       "PDI".CB_FLT_DC24V_K2 := "HDI_CB_FLT_DC24V_K2" XOR "IDI".CB_FLT_DC24V_K2;
       "PDI".CB_FLT_AC400V_K2 := "HDI_CB_FLT_AC400V_K2" XOR "IDI".CB_FLT_AC400V_K2;
       "PDI".SPARE_16_2 := "HDI_SPARE_16_2" XOR "IDI".SPARE_16_2;
       "PDI".CB_FLT_AC230V := "HDI_CB_FLT_AC230V" XOR "IDI".CB_FLT_AC230V;
       "PDI".SPARE_16_4 := "HDI_SPARE_16_4" XOR "IDI".SPARE_16_4;
       "PDI".SPARE_16_5 := "HDI_SPARE_16_5" XOR "IDI".SPARE_16_5;
       "PDI".SPARE_16_6 := "HDI_SPARE_16_6" XOR "IDI".SPARE_16_6;
       "PDI".SPARE_16_7 := "HDI_SPARE_16_7" XOR "IDI".SPARE_16_7;
       "PDI".SPARE_17_0 := "HDI_SPARE_17_0" XOR "IDI".SPARE_17_0;
       "PDI".UPS_24V_ALM := "HDI_UPS_24V_ALM" XOR "IDI".UPS_24V_ALM;
       "PDI".UPS_24V_NRM := "HDI_UPS_24V_NRM" XOR "IDI".UPS_24V_NRM;
       "PDI".EMO := "HDI_EMO" XOR "IDI".EMO;
       "PDI".EMS := "HDI_EMS" XOR "IDI".EMS;
       "PDI".SPARE_17_5 := "HDI_SPARE_17_5" XOR "IDI".SPARE_17_5;
       "PDI".SPARE_17_6 := "HDI_SPARE_17_6" XOR "IDI".SPARE_17_6;
       "PDI".SPARE_17_7 := "HDI_SPARE_17_7" XOR "IDI".SPARE_17_7;
       "PDI".P1_WRN := "HDI_P1_WRN" XOR "IDI".P1_WRN;
       "PDI".P1_FLT := "HDI_P1_FLT" XOR "IDI".P1_FLT;
       "PDI".P1_IS_ON := "HDI_P1_IS_ON" XOR "IDI".P1_IS_ON;
       "PDI".P1_WD := "HDI_P1_WD" XOR "IDI".P1_WD;
       "PDI".FIL_APS := "HDI_FIL_APS" XOR "IDI".FIL_APS;
       "PDI".MON_TMP_P2 := "HDI_MON_TMP_P2" XOR "IDI".MON_TMP_P2;
       "PDI".MON_TMP_P1 := "HDI_MON_TMP_P1" XOR "IDI".MON_TMP_P1;
       "PDI".SPARE_18_7 := "HDI_SPARE_18_7" XOR "IDI".SPARE_18_7;
       "PDI".FCH_LFT_SDL_NUT := "HDI_FCH_LFT_SDL_NUT" XOR "IDI".FCH_LFT_SDL_NUT;
       "PDI".LS_FCH_LFT_DN := "HDI_LS_FCH_LFT_DN" XOR "IDI".LS_FCH_LFT_DN;
       "PDI".LS_FCH_HOOK_WORK := "HDI_LS_FCH_HOOK_WORK" XOR "IDI".LS_FCH_HOOK_WORK;
       "PDI".LS_FCH_HOOK_HOME := "HDI_LS_FCH_HOOK_HOME" XOR "IDI".LS_FCH_HOOK_HOME;
       "PDI".LS_TEC_FLG_DN := "HDI_LS_TEC_FLG_DN" XOR "IDI".LS_TEC_FLG_DN;
       "PDI".TEC_FLG_SDL_NUT := "HDI_TEC_FLG_SDL_NUT" XOR "IDI".TEC_FLG_SDL_NUT;
       "PDI".LS_V11_COV_OP := "HDI_LS_V11_COV_OP" XOR "IDI".LS_V11_COV_OP;
       "PDI".LS_V11_COV_CL := "HDI_LS_V11_COV_CL" XOR "IDI".LS_V11_COV_CL;
       "PDI".GCH_APS := "HDI_GCH_APS" XOR "IDI".GCH_APS;
       "PDI".FCH_APS := "HDI_FCH_APS" XOR "IDI".FCH_APS;
       "PDI".FDR_APS := "HDI_FDR_APS" XOR "IDI".FDR_APS;
       "PDI".FIL_2_APS := "HDI_FIL_2_APS" XOR "IDI".FIL_2_APS;
       "PDI".SPARE_33_4 := "HDI_SPARE_33_4" XOR "IDI".SPARE_33_4;
       "PDI".SPARE_33_5 := "HDI_SPARE_33_5" XOR "IDI".SPARE_33_5;
       "PDI".LS_V2_1_OP := "HDI_LS_V2_1_OP" XOR "IDI".LS_V2_1_OP;
       "PDI".LS_V2_1_CL := "HDI_LS_V2_1_CL" XOR "IDI".LS_V2_1_CL;
       "PDI".CB_FLT_AC400V_K5 := "HDI_CB_FLT_AC400V_K5" XOR "IDI".CB_FLT_AC400V_K5;
       "PDI".CB_FLT_DC24V_K5 := "HDI_CB_FLT_DC24V_K5" XOR "IDI".CB_FLT_DC24V_K5;
       "PDI".LS_MAG_LFT_UP := "HDI_LS_MAG_LFT_UP" XOR "IDI".LS_MAG_LFT_UP;
       "PDI".LS_MAG_LFT_DN := "HDI_LS_MAG_LFT_DN" XOR "IDI".LS_MAG_LFT_DN;
       "PDI".SLS_MAG_LFT := "HDI_SLS_MAG_LFT" XOR "IDI".SLS_MAG_LFT;
       "PDI".MAG_LFT_SDL_NUT1 := "HDI_MAG_LFT_SDL_NUT1" XOR "IDI".MAG_LFT_SDL_NUT1;
       "PDI".MAG_LFT_SDL_NUT2 := "HDI_MAG_LFT_SDL_NUT2" XOR "IDI".MAG_LFT_SDL_NUT2;
       "PDI".MAG_LFT_SDL_NUT3 := "HDI_MAG_LFT_SDL_NUT3" XOR "IDI".MAG_LFT_SDL_NUT3;
       "PDI".OIL_LVL_CR_SFT := "HDI_OIL_LVL_CR_SFT" XOR "IDI".OIL_LVL_CR_SFT;
       "PDI".LS_V1_OP := "HDI_LS_V1_OP" XOR "IDI".LS_V1_OP;
       "PDI".LS_V1_CL := "HDI_LS_V1_CL" XOR "IDI".LS_V1_CL;
       "PDI".MP_ENB_K5 := "HDI_MP_ENB_K5" XOR "IDI".MP_ENB_K5;
       "PDI".SLS_TEC_FLG_LFT := "HDI_SLS_TEC_FLG_LFT" XOR "IDI".SLS_TEC_FLG_LFT;
       "PDI".SLS_FCH_LFT := "HDI_SLS_FCH_LFT" XOR "IDI".SLS_FCH_LFT;
       "PDI".COMP_AIR_OK := "HDI_COMP_AIR_OK" XOR "IDI".COMP_AIR_OK;
       "PDI".COMP_AIR_2_OK := "HDI_COMP_AIR_2_OK" XOR "IDI".COMP_AIR_2_OK;
       "PDI".LS_V1_1_CL := "HDI_LS_V1_1_CL" XOR "IDI".LS_V1_1_CL;
       "PDI".LS_V1_1_OP := "HDI_LS_V1_1_OP" XOR "IDI".LS_V1_1_OP;
       "PDI".LS_V3_4_OP := "HDI_LS_V3_4_OP" XOR "IDI".LS_V3_4_OP;
       "PDI".LS_V3_4_CL := "HDI_LS_V3_4_CL" XOR "IDI".LS_V3_4_CL;
       "PDI".LS_V3_3_OP := "HDI_LS_V3_3_OP" XOR "IDI".LS_V3_3_OP;
       "PDI".LS_V3_3_CL := "HDI_LS_V3_3_CL" XOR "IDI".LS_V3_3_CL;
       "PDI".LS_V2_11_OP := "HDI_LS_V2_11_OP" XOR "IDI".LS_V2_11_OP;
       "PDI".LS_V2_11_CL := "HDI_LS_V2_11_CL" XOR "IDI".LS_V2_11_CL;
       "PDI".ACC_FCH_OV_PRS_1 := "HDI_ACC_FCH_OV_PRS_1" XOR "IDI".ACC_FCH_OV_PRS_1;
       "PDI".ACC_FCH_OV_PRS_2 := "HDI_ACC_FCH_OV_PRS_2" XOR "IDI".ACC_FCH_OV_PRS_2;
       "PDI".SPARE_48_2 := "HDI_SPARE_48_2" XOR "IDI".SPARE_48_2;
       "PDI".ACC_WTR_FLW_OUT_OK := "HDI_ACC_WTR_FLW_OUT_OK" XOR "IDI".ACC_WTR_FLW_OUT_OK;
       "PDI".ACC_WTR_FLW_IN_OK := "HDI_ACC_WTR_FLW_IN_OK" XOR "IDI".ACC_WTR_FLW_IN_OK;
       "PDI".ACC_WTR_TMP_OUT_OK := "HDI_ACC_WTR_TMP_OUT_OK" XOR "IDI".ACC_WTR_TMP_OUT_OK;
       "PDI".OV_PRS_1_FLT := "HDI_OV_PRS_1_FLT" XOR "IDI".OV_PRS_1_FLT;
       "PDI".OV_PRS_2_FLT := "HDI_OV_PRS_2_FLT" XOR "IDI".OV_PRS_2_FLT;
       "PDI".ACC_SC_WTR_OK := "HDI_ACC_SC_WTR_OK" XOR "IDI".ACC_SC_WTR_OK;
       "PDI".ACC_SC_WTR_ATV := "HDI_ACC_SC_WTR_ATV" XOR "IDI".ACC_SC_WTR_ATV;
       "PDI".ACC_SC_HTR_OK := "HDI_ACC_SC_HTR_OK" XOR "IDI".ACC_SC_HTR_OK;
       "PDI".ACC_SC_HTR_ATV := "HDI_ACC_SC_HTR_ATV" XOR "IDI".ACC_SC_HTR_ATV;
       "PDI".ACC_KEY_RST := "HDI_ACC_KEY_RST" XOR "IDI".ACC_KEY_RST;
       "PDI".ACC_CB_FLT_DC24V := "HDI_ACC_CB_FLT_DC24V" XOR "IDI".ACC_CB_FLT_DC24V;
       "PDI".ACC_UPS_24V_ALM := "HDI_ACC_UPS_24V_ALM" XOR "IDI".ACC_UPS_24V_ALM;
       "PDI".ACC_UPS_24V_NRM := "HDI_ACC_UPS_24V_NRM" XOR "IDI".ACC_UPS_24V_NRM;
       "PDI".DPH_RPT_DET_OK := "HDI_DPH_RPT_DET_OK" XOR "IDI".DPH_RPT_DET_OK;
       "PDI".ACC_CB_FLT_AC230V := "HDI_ACC_CB_FLT_AC230V" XOR "IDI".ACC_CB_FLT_AC230V;
       "PDI".SPARE_90_2 := "HDI_SPARE_90_2" XOR "IDI".SPARE_90_2;
       "PDI".SPARE_90_3 := "HDI_SPARE_90_3" XOR "IDI".SPARE_90_3;
       "PDI".SPARE_90_4 := "HDI_SPARE_90_4" XOR "IDI".SPARE_90_4;
       "PDI".SPARE_90_5 := "HDI_SPARE_90_5" XOR "IDI".SPARE_90_5;
       "PDI".SPARE_90_6 := "HDI_SPARE_90_6" XOR "IDI".SPARE_90_6;
       "PDI".SPARE_90_7 := "HDI_SPARE_90_7" XOR "IDI".SPARE_90_7;
       "PDI".FU_P2_RDY := "HDI_FU_P2_RDY" XOR "IDI".FU_P2_RDY;
       "PDI".SPARE_144_1 := "HDI_SPARE_144_1" XOR "IDI".SPARE_144_1;
       "PDI".LS_GCH_UP := "HDI_LS_GCH_UP" XOR "IDI".LS_GCH_UP;
       "PDI".LS_GCH_DN := "HDI_LS_GCH_DN" XOR "IDI".LS_GCH_DN;
       "PDI".LS_GCH_SW_IN := "HDI_LS_GCH_SW_IN" XOR "IDI".LS_GCH_SW_IN;
       "PDI".LS_GCH_SW_CLN := "HDI_LS_GCH_SW_CLN" XOR "IDI".LS_GCH_SW_CLN;
       "PDI".LS_GCH_SW_OUT := "HDI_LS_GCH_SW_OUT" XOR "IDI".LS_GCH_SW_OUT;
       "PDI".LS_GCH_SW_LOCK := "HDI_LS_GCH_SW_LOCK" XOR "IDI".LS_GCH_SW_LOCK;
       "PDI".SLS_GCH_LFT := "HDI_SLS_GCH_LFT" XOR "IDI".SLS_GCH_LFT;
       "PDI".LS_TCH_UP := "HDI_LS_TCH_UP" XOR "IDI".LS_TCH_UP;
       "PDI".LS_TCH_DN := "HDI_LS_TCH_DN" XOR "IDI".LS_TCH_DN;
       "PDI".LS_TCH_SW_IN := "HDI_LS_TCH_SW_IN" XOR "IDI".LS_TCH_SW_IN;
       "PDI".LS_TCH_SW_CLN := "HDI_LS_TCH_SW_CLN" XOR "IDI".LS_TCH_SW_CLN;
       "PDI".LS_TCH_SW_OUT := "HDI_LS_TCH_SW_OUT" XOR "IDI".LS_TCH_SW_OUT;
       "PDI".LS_TCH_SW_LOCK := "HDI_LS_TCH_SW_LOCK" XOR "IDI".LS_TCH_SW_LOCK;
       "PDI".LS_TCH_TILT_0 := "HDI_LS_TCH_TILT_0" XOR "IDI".LS_TCH_TILT_0;
       "PDI".LS_TCH_TILT_30 := "HDI_LS_TCH_TILT_30" XOR "IDI".LS_TCH_TILT_30;
       "PDI".KEY_XT_LFT_SRV := "HDI_KEY_XT_LFT_SRV" XOR "IDI".KEY_XT_LFT_SRV;
       "PDI".LS_V7_UP := "HDI_LS_V7_UP" XOR "IDI".LS_V7_UP;
       "PDI".LS_V7_DN := "HDI_LS_V7_DN" XOR "IDI".LS_V7_DN;
       "PDI".LS_V7_SW_IN := "HDI_LS_V7_SW_IN" XOR "IDI".LS_V7_SW_IN;
       "PDI".LS_V7_SW_OUT := "HDI_LS_V7_SW_OUT" XOR "IDI".LS_V7_SW_OUT;
       "PDI".LS_V7_FLP_OP := "HDI_LS_V7_FLP_OP" XOR "IDI".LS_V7_FLP_OP;
       "PDI".LS_V7_CLN_POS := "HDI_LS_V7_CLN_POS" XOR "IDI".LS_V7_CLN_POS;
       "PDI".LS_GCH_BEL_UP := "HDI_LS_GCH_BEL_UP" XOR "IDI".LS_GCH_BEL_UP;
       "PDI".LS_GCH_BEL_DN := "HDI_LS_GCH_BEL_DN" XOR "IDI".LS_GCH_BEL_DN;
       "PDI".LS_XT_SLID_BW := "HDI_LS_XT_SLID_BW" XOR "IDI".LS_XT_SLID_BW;
       "PDI".LS_XT_SLID_FW := "HDI_LS_XT_SLID_FW" XOR "IDI".LS_XT_SLID_FW;
       "PDI".LS_XT_SLID_MID := "HDI_LS_XT_SLID_MID" XOR "IDI".LS_XT_SLID_MID;
       "PDI".LS_XT_CLP_CON := "HDI_LS_XT_CLP_CON" XOR "IDI".LS_XT_CLP_CON;
       "PDI".LS_XT_TILT_90 := HDI_LS_XT_TILT_90 XOR "IDI".LS_XT_TILT_90;
       "PDI".LS_XT_TILT_75 := HDI_LS_XT_TILT_75 XOR "IDI".LS_XT_TILT_75;
       "PDI".LS_UP_XT_CLP_FLT := "HDI_LS_UP_XT_CLP_FLT" XOR "IDI".LS_UP_XT_CLP_FLT;
       "PDI".SPARE_275_7 := "HDI_SPARE_275_7" XOR "IDI".SPARE_275_7;
       "PDI".LS_UP_XT_CLP_OP := "HDI_LS_UP_XT_CLP_OP" XOR "IDI".LS_UP_XT_CLP_OP;
       "PDI".LS_UP_XT_CLP_CL := "HDI_LS_UP_XT_CLP_CL" XOR "IDI".LS_UP_XT_CLP_CL;
       "PDI".LS_UP_XT_CLP_SAVE := "HDI_LS_UP_XT_CLP_SAVE" XOR "IDI".LS_UP_XT_CLP_SAVE;
       "PDI".LS_UP_XT_CLP_PLATE := "HDI_LS_UP_XT_CLP_PLATE" XOR "IDI".LS_UP_XT_CLP_PLATE;
       "PDI".LS_LO_XT_CLP_FLT := "HDI_LS_LO_XT_CLP_FLT" XOR "IDI".LS_LO_XT_CLP_FLT;
       "PDI".LS_LO_XT_CLP_OP := "HDI_LS_LO_XT_CLP_OP" XOR "IDI".LS_LO_XT_CLP_OP;
       "PDI".LS_LO_XT_CLP_CL := "HDI_LS_LO_XT_CLP_CL" XOR "IDI".LS_LO_XT_CLP_CL;
       "PDI".LS_LO_XT_CLP_SAVE := "HDI_LS_LO_XT_CLP_SAVE" XOR "IDI".LS_LO_XT_CLP_SAVE;
       "PDI".LS_LO_XT_CLP_PLATE := "HDI_LS_LO_XT_CLP_PLATE" XOR "IDI".LS_LO_XT_CLP_PLATE;
       "PDI".LS_HOI_TOOL_INST := "HDI_LS_HOI_TOOL_INST" XOR "IDI".LS_HOI_TOOL_INST;
       "PDI".XT_DRP_OUT_PRT_1_CL := "HDI_XT_DRP_OUT_PRT_1_CL" XOR "IDI".XT_DRP_OUT_PRT_1_CL;
       "PDI".XT_DRP_OUT_PRT_1_OP := "HDI_XT_DRP_OUT_PRT_1_OP" XOR "IDI".XT_DRP_OUT_PRT_1_OP;
       "PDI".XT_DRP_OUT_PRT_2_CL := "HDI_XT_DRP_OUT_PRT_2_CL" XOR "IDI".XT_DRP_OUT_PRT_2_CL;
       "PDI".XT_DRP_OUT_PRT_2_OP := "HDI_XT_DRP_OUT_PRT_2_OP" XOR "IDI".XT_DRP_OUT_PRT_2_OP;
       "PDI".CB_FLT_AC400V_K8 := "HDI_CB_FLT_AC400V_K8" XOR "IDI".CB_FLT_AC400V_K8;
       "PDI".CB_FLT_DC24V_K8 := "HDI_CB_FLT_DC24V_K8" XOR "IDI".CB_FLT_DC24V_K8;
       "PDI".XT_DRP_OUT_PRT_3_CL := "HDI_XT_DRP_OUT_PRT_3_CL" XOR "IDI".XT_DRP_OUT_PRT_3_CL;
       "PDI".XT_DRP_OUT_PRT_3_OP := "HDI_XT_DRP_OUT_PRT_3_OP" XOR "IDI".XT_DRP_OUT_PRT_3_OP;
       "PDI".XT_DRP_OUT_PRT_4_CL := "HDI_XT_DRP_OUT_PRT_4_CL" XOR "IDI".XT_DRP_OUT_PRT_4_CL;
       "PDI".XT_DRP_OUT_PRT_4_OP := "HDI_XT_DRP_OUT_PRT_4_OP" XOR "IDI".XT_DRP_OUT_PRT_4_OP;
       "PDI".LS_XT_HDL_SW_UNLOCK := "HDI_LS_XT_HDL_SW_UNLOCK" XOR "IDI".LS_XT_HDL_SW_UNLOCK;
       "PDI".LS_XT_HDL_SW_LOCK := HDI_LS_XT_HDL_SW_LOCK XOR "IDI".LS_XT_HDL_SW_LOCK;
       "PDI".LS_GCH_DOOR_OP := "HDI_LS_GCH_DOOR_OP" XOR "IDI".LS_GCH_DOOR_OP;
       "PDI".LS_GCH_DOOR_CL := "HDI_LS_GCH_DOOR_CL" XOR "IDI".LS_GCH_DOOR_CL;
       "PDI".MCC_CONTACT_XT := "HDI_MCC_CONTACT_XT" XOR "IDI".MCC_CONTACT_XT;
       "PDI".OIL_LVL_XT_SFT := "HDI_OIL_LVL_XT_SFT" XOR "IDI".OIL_LVL_XT_SFT;
       "PDI".LS_XT_SFT_SRV_POS := "HDI_LS_XT_SFT_SRV_POS" XOR "IDI".LS_XT_SFT_SRV_POS;
       "PDI".LS_XT_TOP_POS := "HDI_LS_XT_TOP_POS" XOR "IDI".LS_XT_TOP_POS;
       "PDI".SLS_TCH_LFT := "HDI_SLS_TCH_LFT" XOR "IDI".SLS_TCH_LFT;
       "PDI".XT_ROT_CAM_TRG := "HDI_XT_ROT_CAM_TRG" XOR "IDI".XT_ROT_CAM_TRG;
       "PDI".MP_ENB_K8 := "HDI_MP_ENB_K8" XOR "IDI".MP_ENB_K8;
       "PDI".MP_ENB_K9 := "HDI_MP_ENB_K9" XOR "IDI".MP_ENB_K9;
       "PDI".LS_V3_OP := "HDI_LS_V3_OP" XOR "IDI".LS_V3_OP;
       "PDI".LS_V3_CL := "HDI_LS_V3_CL" XOR "IDI".LS_V3_CL;
       "PDI".FDR_LS_V3_2_OP := "HDI_FDR_LS_V3_2_OP" XOR "IDI".FDR_LS_V3_2_OP;
       "PDI".FDR_LS_V3_2_CL := "HDI_FDR_LS_V3_2_CL" XOR "IDI".FDR_LS_V3_2_CL;
       "PDI".LSR_SEN_OBJ_DET := "HDI_LSR_SEN_OBJ_DET" XOR "IDI".LSR_SEN_OBJ_DET;
       "PDI".SPARE_280_5 := "HDI_SPARE_280_5" XOR "IDI".SPARE_280_5;
       "PDI".SPARE_280_6 := "HDI_SPARE_280_6" XOR "IDI".SPARE_280_6;
       "PDI".SPARE_280_7 := "HDI_SPARE_280_7" XOR "IDI".SPARE_280_7;
       "PDI".LS_V11_OP := "HDI_LS_V11_OP" XOR "IDI".LS_V11_OP;
       "PDI".LS_V11_CL := "HDI_LS_V11_CL" XOR "IDI".LS_V11_CL;
       "PDI".FDR_HOP_CON := "HDI_FDR_HOP_CON" XOR "IDI".FDR_HOP_CON;
   END_IF;
END_FUNCTION_BLOCK

FUNCTION_BLOCK "PM_DO"   // FB18, SCL
{ S7_Optimized_Access := 'FALSE' }
VERSION : 0.0
// --------------------------------------------------------------------------------
//     program:         PM_DO
//     description :    automatically generated PM_DO
//     name:            hp
//     date        :    03.02.2021
// 
//     revision:
//     name:
//     Date:
//                     (c)CGS
//     --------------------------------------------------------------------------------
   VAR
      y : Bool;
      count : Int := 8;
   END_VAR
   VAR_TEMP
      x : Bool;
   END_VAR
BEGIN


   IF "SY".SRM_ON THEN

       "HDO_HOR_OPP_K2" := "SDO".HOR_OPP_K2 XOR "IDO".HOR_OPP_K2;
       "HDO_LMP_RD_K2" := "SDO".LMP_RD_K2 XOR "IDO".LMP_RD_K2;
       "HDO_LMP_YE_K2" := "SDO".LMP_YE_K2 XOR "IDO".LMP_YE_K2;
       "HDO_LMP_GN_K2" := "SDO".LMP_GN_K2 XOR "IDO".LMP_GN_K2;
       "HDO_LMP_BU_K2" := "SDO".LMP_BU_K2 XOR "IDO".LMP_BU_K2;
       "HDO_HOR_MAG_ACTIVE" := "SDO".HOR_MAG_ACTIVE XOR "IDO".HOR_MAG_ACTIVE;
       "HDO_LMP_MAG_ACTIVE" := "SDO".LMP_MAG_ACTIVE XOR "IDO".LMP_MAG_ACTIVE;
       "HDO_SPARE_16_7" := "SDO".SPARE_16_7 XOR "IDO".SPARE_16_7;
       "HDO_P1_ON" := "SDO".P1_ON XOR "IDO".P1_ON;
       "HDO_P3_ON" := "SDO".P3_ON XOR "IDO".P3_ON;
       "HDO_P2_ON" := "SDO".P2_ON XOR "IDO".P2_ON;
       "HDO_P1_SEAL_GAS" := "SDO".P1_SEAL_GAS XOR "IDO".P1_SEAL_GAS;
       "HDO_P3_SEAL_GAS" := "SDO".P3_SEAL_GAS XOR "IDO".P3_SEAL_GAS;
       "HDO_HTR_PWR_ON" := "SDO".HTR_PWR_ON XOR "IDO".HTR_PWR_ON;
       "HDO_V10" := "SDO".V10 XOR "IDO".V10;
       "HDO_MON_TMP_P2_RES" := "SDO".MON_TMP_P2_RES XOR "IDO".MON_TMP_P2_RES;
       "HDO_SPARE_18_0" := "SDO".SPARE_18_0 XOR "IDO".SPARE_18_0;
       "HDO_SPARE_18_1" := "SDO".SPARE_18_1 XOR "IDO".SPARE_18_1;
       "HDO_SPARE_18_2" := "SDO".SPARE_18_2 XOR "IDO".SPARE_18_2;
       "HDO_SPARE_18_3" := "SDO".SPARE_18_3 XOR "IDO".SPARE_18_3;
       "HDO_SPARE_18_4" := "SDO".SPARE_18_4 XOR "IDO".SPARE_18_4;
       "HDO_SPARE_18_5" := "SDO".SPARE_18_5 XOR "IDO".SPARE_18_5;
       "HDO_SPARE_18_6" := "SDO".SPARE_18_6 XOR "IDO".SPARE_18_6;
       "HDO_SPARE_18_7" := "SDO".SPARE_18_7 XOR "IDO".SPARE_18_7;
       "HDO_V1_OP" := "SDO".V1_OP XOR "IDO".V1_OP;
       "HDO_V1_CL" := "SDO".V1_CL XOR "IDO".V1_CL;
       "HDO_SPARE_32_2" := "SDO".SPARE_32_2 XOR "IDO".SPARE_32_2;
       "HDO_SPARE_32_3" := "SDO".SPARE_32_3 XOR "IDO".SPARE_32_3;
       "HDO_SPARE_32_4" := "SDO".SPARE_32_4 XOR "IDO".SPARE_32_4;
       "HDO_CR_ROT_ENB" := "SDO".CR_ROT_ENB XOR "IDO".CR_ROT_ENB;
       "HDO_CR_LFT_ENB" := "SDO".CR_LFT_ENB XOR "IDO".CR_LFT_ENB;
       "HDO_FU_FCB_HDL_ON" := "SDO".FU_FCB_HDL_ON XOR "IDO".FU_FCB_HDL_ON;
       "HDO_TEC_FLG_LFT_ENB" := "SDO".TEC_FLG_LFT_ENB XOR "IDO".TEC_FLG_LFT_ENB;
       "HDO_FCH_LFT_ENB" := "SDO".FCH_LFT_ENB XOR "IDO".FCH_LFT_ENB;
       "HDO_MAG_LFT_UP" := "SDO".MAG_LFT_UP XOR "IDO".MAG_LFT_UP;
       "HDO_MAG_LFT_DN" := "SDO".MAG_LFT_DN XOR "IDO".MAG_LFT_DN;
       "HDO_BRK_MAG_LFT" := "SDO".BRK_MAG_LFT XOR "IDO".BRK_MAG_LFT;
       "HDO_SPARE_33_5" := "SDO".SPARE_33_5 XOR "IDO".SPARE_33_5;
       "HDO_SPARE_33_6" := "SDO".SPARE_33_6 XOR "IDO".SPARE_33_6;
       "HDO_SPARE_33_7" := "SDO".SPARE_33_7 XOR "IDO".SPARE_33_7;
       "HDO_V1_1_OP" := "SDO".V1_1_OP XOR "IDO".V1_1_OP;
       "HDO_V1_1_CL" := "SDO".V1_1_CL XOR "IDO".V1_1_CL;
       "HDO_SPARE_34_2" := "SDO".SPARE_34_2 XOR "IDO".SPARE_34_2;
       "HDO_SPARE_34_3" := "SDO".SPARE_34_3 XOR "IDO".SPARE_34_3;
       "HDO_SPARE_34_4" := "SDO".SPARE_34_4 XOR "IDO".SPARE_34_4;
       "HDO_SPARE_34_5" := "SDO".SPARE_34_5 XOR "IDO".SPARE_34_5;
       "HDO_SPARE_34_6" := "SDO".SPARE_34_6 XOR "IDO".SPARE_34_6;
       "HDO_SPARE_34_7" := "SDO".SPARE_34_7 XOR "IDO".SPARE_34_7;
       "HDO_ACC_SC_HTR_STR" := "SDO".ACC_SC_HTR_STR XOR "IDO".ACC_SC_HTR_STR;
       "HDO_ACC_SC_HTR_RST" := "SDO".ACC_SC_HTR_RST XOR "IDO".ACC_SC_HTR_RST;
       "HDO_ACC_SC_WTR_STR" := "SDO".ACC_SC_WTR_STR XOR "IDO".ACC_SC_WTR_STR;
       "HDO_ACC_SC_WTR_RST" := "SDO".ACC_SC_WTR_RST XOR "IDO".ACC_SC_WTR_RST;
       "HDO_ACC_ALM_LT_1" := "SDO".ACC_ALM_LT_1 XOR "IDO".ACC_ALM_LT_1;
       "HDO_ACC_ALM_SND_1" := "SDO".ACC_ALM_SND_1 XOR "IDO".ACC_ALM_SND_1;
       "HDO_ACC_ALM_LT_2" := "SDO".ACC_ALM_LT_2 XOR "IDO".ACC_ALM_LT_2;
       "HDO_ACC_ALM_SND_2" := "SDO".ACC_ALM_SND_2 XOR "IDO".ACC_ALM_SND_2;
       "HDO_FCH_HOOK_HOME" := "SDO".FCH_HOOK_HOME XOR "IDO".FCH_HOOK_HOME;
       "HDO_FCH_HOOK_WORK" := "SDO".FCH_HOOK_WORK XOR "IDO".FCH_HOOK_WORK;
       "HDO_UP_FCH_SW_BRK" := "SDO".UP_FCH_SW_BRK XOR "IDO".UP_FCH_SW_BRK;
       "HDO_LO_FCH_SW_BRK" := "SDO".LO_FCH_SW_BRK XOR "IDO".LO_FCH_SW_BRK;
       "HDO_TEC_FLG_SW_BRK" := "SDO".TEC_FLG_SW_BRK XOR "IDO".TEC_FLG_SW_BRK;
       "HDO_V25" := "SDO".V25 XOR "IDO".V25;
       "HDO_V2_1" := "SDO".V2_1 XOR "IDO".V2_1;
       "HDO_V21" := "SDO".V21 XOR "IDO".V21;
       "HDO_V19" := "SDO".V19 XOR "IDO".V19;
       "HDO_V20" := "SDO".V20 XOR "IDO".V20;
       "HDO_V22" := "SDO".V22 XOR "IDO".V22;
       "HDO_V9_2" := "SDO".V9_2 XOR "IDO".V9_2;
       "HDO_V22_1" := "SDO".V22_1 XOR "IDO".V22_1;
       "HDO_V3_4" := "SDO".V3_4 XOR "IDO".V3_4;
       "HDO_V3_3" := "SDO".V3_3 XOR "IDO".V3_3;
       "HDO_V2_11" := "SDO".V2_11 XOR "IDO".V2_11;
       "HDO_P2_FU_ON" := "SDO".P2_FU_ON XOR "IDO".P2_FU_ON;
       "HDO_P2_FU_RES" := "SDO".P2_FU_RES XOR "IDO".P2_FU_RES;
       "HDO_V4" := "SDO".V4 XOR "IDO".V4;
       "HDO_V5" := "SDO".V5 XOR "IDO".V5;
       "HDO_V6" := "SDO".V6 XOR "IDO".V6;
       "HDO_V3" := "SDO".V3 XOR "IDO".V3;
       "HDO_V3_2" := "SDO".V3_2 XOR "IDO".V3_2;
       "HDO_V24" := "SDO".V24 XOR "IDO".V24;
       "HDO_XT_DRP_OUT_PRT_CL" := "SDO".XT_DRP_OUT_PRT_CL XOR "IDO".XT_DRP_OUT_PRT_CL;
       "HDO_XT_DRP_OUT_PRT_OP" := "SDO".XT_DRP_OUT_PRT_OP XOR "IDO".XT_DRP_OUT_PRT_OP;
       "HDO_TCH_SW_LOCK" := "SDO".TCH_SW_LOCK XOR "IDO".TCH_SW_LOCK;
       "HDO_TCH_SW_UNLOCK" := "SDO".TCH_SW_UNLOCK XOR "IDO".TCH_SW_UNLOCK;
       "HDO_GCH_SW_LOCK" := "SDO".GCH_SW_LOCK XOR "IDO".GCH_SW_LOCK;
       "HDO_GCH_SW_UNLOCK" := "SDO".GCH_SW_UNLOCK XOR "IDO".GCH_SW_UNLOCK;
       "HDO_XT_HDL_SW_LOCK" := "SDO".XT_HDL_SW_LOCK XOR "IDO".XT_HDL_SW_LOCK;
       "HDO_XT_HDL_SW_UNLOCK" := "SDO".XT_HDL_SW_UNLOCK XOR "IDO".XT_HDL_SW_UNLOCK;
       "HDO_FDR_V11_OP" := "SDO".FDR_V11_OP XOR "IDO".FDR_V11_OP;
       "HDO_FDR_V11_CL" := "SDO".FDR_V11_CL XOR "IDO".FDR_V11_CL;
       "HDO_FDR_V11_CVR_OP" := "SDO".FDR_V11_CVR_OP XOR "IDO".FDR_V11_CVR_OP;
       "HDO_FDR_V11_CVR_CL" := "SDO".FDR_V11_CVR_CL XOR "IDO".FDR_V11_CVR_CL;
       "HDO_SPARE_226_2" := "SDO".SPARE_226_2 XOR "IDO".SPARE_226_2;
       "HDO_SPARE_226_3" := "SDO".SPARE_226_3 XOR "IDO".SPARE_226_3;
       "HDO_SPARE_226_4" := "SDO".SPARE_226_4 XOR "IDO".SPARE_226_4;
       "HDO_SPARE_226_5" := "SDO".SPARE_226_5 XOR "IDO".SPARE_226_5;
       "HDO_SPARE_226_6" := "SDO".SPARE_226_6 XOR "IDO".SPARE_226_6;
       "HDO_SPARE_226_7" := "SDO".SPARE_226_7 XOR "IDO".SPARE_226_7;
       "HDO_HOR_OPP_K8" := "SDO".HOR_OPP_K8 XOR "IDO".HOR_OPP_K8;
       "HDO_LMP_RD_K8" := "SDO".LMP_RD_K8 XOR "IDO".LMP_RD_K8;
       "HDO_LMP_YE_K8" := "SDO".LMP_YE_K8 XOR "IDO".LMP_YE_K8;
       "HDO_LMP_GN_K8" := "SDO".LMP_GN_K8 XOR "IDO".LMP_GN_K8;
       "HDO_LMP_BU_K8" := "SDO".LMP_BU_K8 XOR "IDO".LMP_BU_K8;
       "HDO_XT_ROT_ENB" := "SDO".XT_ROT_ENB XOR "IDO".XT_ROT_ENB;
       "HDO_XT_LFT_ENB" := "SDO".XT_LFT_ENB XOR "IDO".XT_LFT_ENB;
       "HDO_XT_HDL_LFT_ENB" := "SDO".XT_HDL_LFT_ENB XOR "IDO".XT_HDL_LFT_ENB;
       "HDO_XT_HDL_SW_ENB" := "SDO".XT_HDL_SW_ENB XOR "IDO".XT_HDL_SW_ENB;
       "HDO_FU_GCB_HDL_ON" := "SDO".FU_GCB_HDL_ON XOR "IDO".FU_GCB_HDL_ON;
       "HDO_LSR_SEN_PWR_ON" := "SDO".LSR_SEN_PWR_ON XOR "IDO".LSR_SEN_PWR_ON;
       "HDO_SPARE_273_3" := "SDO".SPARE_273_3 XOR "IDO".SPARE_273_3;
       "HDO_SPARE_273_4" := "SDO".SPARE_273_4 XOR "IDO".SPARE_273_4;
       "HDO_SPARE_273_5" := "SDO".SPARE_273_5 XOR "IDO".SPARE_273_5;
       "HDO_XT_HDL_SLID_FW" := "SDO".XT_HDL_SLID_FW XOR "IDO".XT_HDL_SLID_FW;
       "HDO_XT_HDL_SLID_BW" := "SDO".XT_HDL_SLID_BW XOR "IDO".XT_HDL_SLID_BW;
       "HDO_XT_CLP_TILT_BW" := "SDO".XT_CLP_TILT_BW XOR "IDO".XT_CLP_TILT_BW;
       "HDO_XT_CLP_TILT_FW" := "SDO".XT_CLP_TILT_FW XOR "IDO".XT_CLP_TILT_FW;
       "HDO_XT_CLP_TILT_BRK" := "SDO".XT_CLP_TILT_BRK XOR "IDO".XT_CLP_TILT_BRK;
       "HDO_XT_CLP_ABV_OP" := "SDO".XT_CLP_ABV_OP XOR "IDO".XT_CLP_ABV_OP;
       "HDO_XT_CLP_ABV_CL" := "SDO".XT_CLP_ABV_CL XOR "IDO".XT_CLP_ABV_CL;
       "HDO_XT_CLP_ABV_BRK" := "SDO".XT_CLP_ABV_BRK XOR "IDO".XT_CLP_ABV_BRK;
       "HDO_XT_CLP_ABV_RST" := "SDO".XT_CLP_ABV_RST XOR "IDO".XT_CLP_ABV_RST;
       "HDO_GCH_LFT_ENB" := "SDO".GCH_LFT_ENB XOR "IDO".GCH_LFT_ENB;
       "HDO_XT_CLP_BLW_OP" := "SDO".XT_CLP_BLW_OP XOR "IDO".XT_CLP_BLW_OP;
       "HDO_XT_CLP_BLW_CL" := "SDO".XT_CLP_BLW_CL XOR "IDO".XT_CLP_BLW_CL;
       "HDO_XT_CLP_BLW_BRK" := "SDO".XT_CLP_BLW_BRK XOR "IDO".XT_CLP_BLW_BRK;
       "HDO_XT_CLP_BLW_RST" := "SDO".XT_CLP_BLW_RST XOR "IDO".XT_CLP_BLW_RST;
       "HDO_MCC_TEST_XT" := "SDO".MCC_TEST_XT XOR "IDO".MCC_TEST_XT;
       "HDO_MCC_ENB_XT" := "SDO".MCC_ENB_XT XOR "IDO".MCC_ENB_XT;
       "HDO_TCH_LFT_ENB" := "SDO".TCH_LFT_ENB XOR "IDO".TCH_LFT_ENB;
       "HDO_TCH_TILT_ENB" := "SDO".TCH_TILT_ENB XOR "IDO".TCH_TILT_ENB;
       "HDO_GTE_V_LFT_ENB" := "SDO".GTE_V_LFT_ENB XOR "IDO".GTE_V_LFT_ENB;
       "HDO_GTE_V_SW_ENB" := "SDO".GTE_V_SW_ENB XOR "IDO".GTE_V_SW_ENB;
       "HDO_BEL_LFT_ENB" := "SDO".BEL_LFT_ENB XOR "IDO".BEL_LFT_ENB;
       "HDO_HOR_OPP_K9" := "SDO".HOR_OPP_K9 XOR "IDO".HOR_OPP_K9;
       "HDO_LMP_RD_K9" := "SDO".LMP_RD_K9 XOR "IDO".LMP_RD_K9;
       "HDO_LMP_YE_K9" := "SDO".LMP_YE_K9 XOR "IDO".LMP_YE_K9;
       "HDO_LMP_GN_K9" := "SDO".LMP_GN_K9 XOR "IDO".LMP_GN_K9;
       "HDO_LMP_BU_K9" := "SDO".LMP_BU_K9 XOR "IDO".LMP_BU_K9;
   ELSE
       IF NOT "SY".SIM_ON THEN

           "HDO_HOR_OPP_K2" := "PDO".HOR_OPP_K2 XOR "IDO".HOR_OPP_K2;
           "HDO_LMP_RD_K2" := "PDO".LMP_RD_K2 XOR "IDO".LMP_RD_K2;
           "HDO_LMP_YE_K2" := "PDO".LMP_YE_K2 XOR "IDO".LMP_YE_K2;
           "HDO_LMP_GN_K2" := "PDO".LMP_GN_K2 XOR "IDO".LMP_GN_K2;
           "HDO_LMP_BU_K2" := "PDO".LMP_BU_K2 XOR "IDO".LMP_BU_K2;
           "HDO_HOR_MAG_ACTIVE" := "PDO".HOR_MAG_ACTIVE XOR "IDO".HOR_MAG_ACTIVE;
           "HDO_LMP_MAG_ACTIVE" := "PDO".LMP_MAG_ACTIVE XOR "IDO".LMP_MAG_ACTIVE;
           "HDO_SPARE_16_7" := "PDO".SPARE_16_7 XOR "IDO".SPARE_16_7;
           "HDO_P1_ON" := "PDO".P1_ON XOR "IDO".P1_ON;
           "HDO_P3_ON" := "PDO".P3_ON XOR "IDO".P3_ON;
           "HDO_P2_ON" := "PDO".P2_ON XOR "IDO".P2_ON;
           "HDO_P1_SEAL_GAS" := "PDO".P1_SEAL_GAS XOR "IDO".P1_SEAL_GAS;
           "HDO_P3_SEAL_GAS" := "PDO".P3_SEAL_GAS XOR "IDO".P3_SEAL_GAS;
           "HDO_HTR_PWR_ON" := "PDO".HTR_PWR_ON XOR "IDO".HTR_PWR_ON;
           "HDO_V10" := "PDO".V10 XOR "IDO".V10;
           "HDO_MON_TMP_P2_RES" := "PDO".MON_TMP_P2_RES XOR "IDO".MON_TMP_P2_RES;
           "HDO_SPARE_18_0" := "PDO".SPARE_18_0 XOR "IDO".SPARE_18_0;
           "HDO_SPARE_18_1" := "PDO".SPARE_18_1 XOR "IDO".SPARE_18_1;
           "HDO_SPARE_18_2" := "PDO".SPARE_18_2 XOR "IDO".SPARE_18_2;
           "HDO_SPARE_18_3" := "PDO".SPARE_18_3 XOR "IDO".SPARE_18_3;
           "HDO_SPARE_18_4" := "PDO".SPARE_18_4 XOR "IDO".SPARE_18_4;
           "HDO_SPARE_18_5" := "PDO".SPARE_18_5 XOR "IDO".SPARE_18_5;
           "HDO_SPARE_18_6" := "PDO".SPARE_18_6 XOR "IDO".SPARE_18_6;
           "HDO_SPARE_18_7" := "PDO".SPARE_18_7 XOR "IDO".SPARE_18_7;
           "HDO_V1_OP" := "PDO".V1_OP XOR "IDO".V1_OP;
           "HDO_V1_CL" := "PDO".V1_CL XOR "IDO".V1_CL;
           "HDO_SPARE_32_2" := "PDO".SPARE_32_2 XOR "IDO".SPARE_32_2;
           "HDO_SPARE_32_3" := "PDO".SPARE_32_3 XOR "IDO".SPARE_32_3;
           "HDO_SPARE_32_4" := "PDO".SPARE_32_4 XOR "IDO".SPARE_32_4;
           "HDO_CR_ROT_ENB" := "PDO".CR_ROT_ENB XOR "IDO".CR_ROT_ENB;
           "HDO_CR_LFT_ENB" := "PDO".CR_LFT_ENB XOR "IDO".CR_LFT_ENB;
           "HDO_FU_FCB_HDL_ON" := "PDO".FU_FCB_HDL_ON XOR "IDO".FU_FCB_HDL_ON;
           "HDO_TEC_FLG_LFT_ENB" := "PDO".TEC_FLG_LFT_ENB XOR "IDO".TEC_FLG_LFT_ENB;
           "HDO_FCH_LFT_ENB" := "PDO".FCH_LFT_ENB XOR "IDO".FCH_LFT_ENB;
           "HDO_MAG_LFT_UP" := "PDO".MAG_LFT_UP XOR "IDO".MAG_LFT_UP;
           "HDO_MAG_LFT_DN" := "PDO".MAG_LFT_DN XOR "IDO".MAG_LFT_DN;
           "HDO_BRK_MAG_LFT" := "PDO".BRK_MAG_LFT XOR "IDO".BRK_MAG_LFT;
           "HDO_SPARE_33_5" := "PDO".SPARE_33_5 XOR "IDO".SPARE_33_5;
           "HDO_SPARE_33_6" := "PDO".SPARE_33_6 XOR "IDO".SPARE_33_6;
           "HDO_SPARE_33_7" := "PDO".SPARE_33_7 XOR "IDO".SPARE_33_7;
           "HDO_V1_1_OP" := "PDO".V1_1_OP XOR "IDO".V1_1_OP;
           "HDO_V1_1_CL" := "PDO".V1_1_CL XOR "IDO".V1_1_CL;
           "HDO_SPARE_34_2" := "PDO".SPARE_34_2 XOR "IDO".SPARE_34_2;
           "HDO_SPARE_34_3" := "PDO".SPARE_34_3 XOR "IDO".SPARE_34_3;
           "HDO_SPARE_34_4" := "PDO".SPARE_34_4 XOR "IDO".SPARE_34_4;
           "HDO_SPARE_34_5" := "PDO".SPARE_34_5 XOR "IDO".SPARE_34_5;
           "HDO_SPARE_34_6" := "PDO".SPARE_34_6 XOR "IDO".SPARE_34_6;
           "HDO_SPARE_34_7" := "PDO".SPARE_34_7 XOR "IDO".SPARE_34_7;
           "HDO_ACC_SC_HTR_STR" := "PDO".ACC_SC_HTR_STR XOR "IDO".ACC_SC_HTR_STR;
           "HDO_ACC_SC_HTR_RST" := "PDO".ACC_SC_HTR_RST XOR "IDO".ACC_SC_HTR_RST;
           "HDO_ACC_SC_WTR_STR" := "PDO".ACC_SC_WTR_STR XOR "IDO".ACC_SC_WTR_STR;
           "HDO_ACC_SC_WTR_RST" := "PDO".ACC_SC_WTR_RST XOR "IDO".ACC_SC_WTR_RST;
           "HDO_ACC_ALM_LT_1" := "PDO".ACC_ALM_LT_1 XOR "IDO".ACC_ALM_LT_1;
           "HDO_ACC_ALM_SND_1" := "PDO".ACC_ALM_SND_1 XOR "IDO".ACC_ALM_SND_1;
           "HDO_ACC_ALM_LT_2" := "PDO".ACC_ALM_LT_2 XOR "IDO".ACC_ALM_LT_2;
           "HDO_ACC_ALM_SND_2" := "PDO".ACC_ALM_SND_2 XOR "IDO".ACC_ALM_SND_2;
           "HDO_FCH_HOOK_HOME" := "PDO".FCH_HOOK_HOME XOR "IDO".FCH_HOOK_HOME;
           "HDO_FCH_HOOK_WORK" := "PDO".FCH_HOOK_WORK XOR "IDO".FCH_HOOK_WORK;
           "HDO_UP_FCH_SW_BRK" := "PDO".UP_FCH_SW_BRK XOR "IDO".UP_FCH_SW_BRK;
           "HDO_LO_FCH_SW_BRK" := "PDO".LO_FCH_SW_BRK XOR "IDO".LO_FCH_SW_BRK;
           "HDO_TEC_FLG_SW_BRK" := "PDO".TEC_FLG_SW_BRK XOR "IDO".TEC_FLG_SW_BRK;
           "HDO_V25" := "PDO".V25 XOR "IDO".V25;
           "HDO_V2_1" := "PDO".V2_1 XOR "IDO".V2_1;
           "HDO_V21" := "PDO".V21 XOR "IDO".V21;
           "HDO_V19" := "PDO".V19 XOR "IDO".V19;
           "HDO_V20" := "PDO".V20 XOR "IDO".V20;
           "HDO_V22" := "PDO".V22 XOR "IDO".V22;
           "HDO_V9_2" := "PDO".V9_2 XOR "IDO".V9_2;
           "HDO_V22_1" := "PDO".V22_1 XOR "IDO".V22_1;
           "HDO_V3_4" := "PDO".V3_4 XOR "IDO".V3_4;
           "HDO_V3_3" := "PDO".V3_3 XOR "IDO".V3_3;
           "HDO_V2_11" := "PDO".V2_11 XOR "IDO".V2_11;
           "HDO_P2_FU_ON" := "PDO".P2_FU_ON XOR "IDO".P2_FU_ON;
           "HDO_P2_FU_RES" := "PDO".P2_FU_RES XOR "IDO".P2_FU_RES;
           "HDO_V4" := "PDO".V4 XOR "IDO".V4;
           "HDO_V5" := "PDO".V5 XOR "IDO".V5;
           "HDO_V6" := "PDO".V6 XOR "IDO".V6;
           "HDO_V3" := "PDO".V3 XOR "IDO".V3;
           "HDO_V3_2" := "PDO".V3_2 XOR "IDO".V3_2;
           "HDO_V24" := "PDO".V24 XOR "IDO".V24;
           "HDO_XT_DRP_OUT_PRT_CL" := "PDO".XT_DRP_OUT_PRT_CL XOR "IDO".XT_DRP_OUT_PRT_CL;
           "HDO_XT_DRP_OUT_PRT_OP" := "PDO".XT_DRP_OUT_PRT_OP XOR "IDO".XT_DRP_OUT_PRT_OP;
           "HDO_TCH_SW_LOCK" := "PDO".TCH_SW_LOCK XOR "IDO".TCH_SW_LOCK;
           "HDO_TCH_SW_UNLOCK" := "PDO".TCH_SW_UNLOCK XOR "IDO".TCH_SW_UNLOCK;
           "HDO_GCH_SW_LOCK" := "PDO".GCH_SW_LOCK XOR "IDO".GCH_SW_LOCK;
           "HDO_GCH_SW_UNLOCK" := "PDO".GCH_SW_UNLOCK XOR "IDO".GCH_SW_UNLOCK;
           "HDO_XT_HDL_SW_LOCK" := "PDO".XT_HDL_SW_LOCK XOR "IDO".XT_HDL_SW_LOCK;
           "HDO_XT_HDL_SW_UNLOCK" := "PDO".XT_HDL_SW_UNLOCK XOR "IDO".XT_HDL_SW_UNLOCK;
           "HDO_FDR_V11_OP" := "PDO".FDR_V11_OP XOR "IDO".FDR_V11_OP;
           "HDO_FDR_V11_CL" := "PDO".FDR_V11_CL XOR "IDO".FDR_V11_CL;
           "HDO_FDR_V11_CVR_OP" := "PDO".FDR_V11_CVR_OP XOR "IDO".FDR_V11_CVR_OP;
           "HDO_FDR_V11_CVR_CL" := "PDO".FDR_V11_CVR_CL XOR "IDO".FDR_V11_CVR_CL;
           "HDO_SPARE_226_2" := "PDO".SPARE_226_2 XOR "IDO".SPARE_226_2;
           "HDO_SPARE_226_3" := "PDO".SPARE_226_3 XOR "IDO".SPARE_226_3;
           "HDO_SPARE_226_4" := "PDO".SPARE_226_4 XOR "IDO".SPARE_226_4;
           "HDO_SPARE_226_5" := "PDO".SPARE_226_5 XOR "IDO".SPARE_226_5;
           "HDO_SPARE_226_6" := "PDO".SPARE_226_6 XOR "IDO".SPARE_226_6;
           "HDO_SPARE_226_7" := "PDO".SPARE_226_7 XOR "IDO".SPARE_226_7;
           "HDO_HOR_OPP_K8" := "PDO".HOR_OPP_K8 XOR "IDO".HOR_OPP_K8;
           "HDO_LMP_RD_K8" := "PDO".LMP_RD_K8 XOR "IDO".LMP_RD_K8;
           "HDO_LMP_YE_K8" := "PDO".LMP_YE_K8 XOR "IDO".LMP_YE_K8;
           "HDO_LMP_GN_K8" := "PDO".LMP_GN_K8 XOR "IDO".LMP_GN_K8;
           "HDO_LMP_BU_K8" := "PDO".LMP_BU_K8 XOR "IDO".LMP_BU_K8;
           "HDO_XT_ROT_ENB" := "PDO".XT_ROT_ENB XOR "IDO".XT_ROT_ENB;
           "HDO_XT_LFT_ENB" := "PDO".XT_LFT_ENB XOR "IDO".XT_LFT_ENB;
           "HDO_XT_HDL_LFT_ENB" := "PDO".XT_HDL_LFT_ENB XOR "IDO".XT_HDL_LFT_ENB;
           "HDO_XT_HDL_SW_ENB" := "PDO".XT_HDL_SW_ENB XOR "IDO".XT_HDL_SW_ENB;
           "HDO_FU_GCB_HDL_ON" := "PDO".FU_GCB_HDL_ON XOR "IDO".FU_GCB_HDL_ON;
           "HDO_LSR_SEN_PWR_ON" := "PDO".LSR_SEN_PWR_ON XOR "IDO".LSR_SEN_PWR_ON;
           "HDO_SPARE_273_3" := "PDO".SPARE_273_3 XOR "IDO".SPARE_273_3;
           "HDO_SPARE_273_4" := "PDO".SPARE_273_4 XOR "IDO".SPARE_273_4;
           "HDO_SPARE_273_5" := "PDO".SPARE_273_5 XOR "IDO".SPARE_273_5;
           "HDO_XT_HDL_SLID_FW" := "PDO".XT_HDL_SLID_FW XOR "IDO".XT_HDL_SLID_FW;
           "HDO_XT_HDL_SLID_BW" := "PDO".XT_HDL_SLID_BW XOR "IDO".XT_HDL_SLID_BW;
           "HDO_XT_CLP_TILT_BW" := "PDO".XT_CLP_TILT_BW XOR "IDO".XT_CLP_TILT_BW;
           "HDO_XT_CLP_TILT_FW" := "PDO".XT_CLP_TILT_FW XOR "IDO".XT_CLP_TILT_FW;
           "HDO_XT_CLP_TILT_BRK" := "PDO".XT_CLP_TILT_BRK XOR "IDO".XT_CLP_TILT_BRK;
           "HDO_XT_CLP_ABV_OP" := "PDO".XT_CLP_ABV_OP XOR "IDO".XT_CLP_ABV_OP;
           "HDO_XT_CLP_ABV_CL" := "PDO".XT_CLP_ABV_CL XOR "IDO".XT_CLP_ABV_CL;
           "HDO_XT_CLP_ABV_BRK" := "PDO".XT_CLP_ABV_BRK XOR "IDO".XT_CLP_ABV_BRK;
           "HDO_XT_CLP_ABV_RST" := "PDO".XT_CLP_ABV_RST XOR "IDO".XT_CLP_ABV_RST;
           "HDO_GCH_LFT_ENB" := "PDO".GCH_LFT_ENB XOR "IDO".GCH_LFT_ENB;
           "HDO_XT_CLP_BLW_OP" := "PDO".XT_CLP_BLW_OP XOR "IDO".XT_CLP_BLW_OP;
           "HDO_XT_CLP_BLW_CL" := "PDO".XT_CLP_BLW_CL XOR "IDO".XT_CLP_BLW_CL;
           "HDO_XT_CLP_BLW_BRK" := "PDO".XT_CLP_BLW_BRK XOR "IDO".XT_CLP_BLW_BRK;
           "HDO_XT_CLP_BLW_RST" := "PDO".XT_CLP_BLW_RST XOR "IDO".XT_CLP_BLW_RST;
           "HDO_MCC_TEST_XT" := "PDO".MCC_TEST_XT XOR "IDO".MCC_TEST_XT;
           "HDO_MCC_ENB_XT" := "PDO".MCC_ENB_XT XOR "IDO".MCC_ENB_XT;
           "HDO_TCH_LFT_ENB" := "PDO".TCH_LFT_ENB XOR "IDO".TCH_LFT_ENB;
           "HDO_TCH_TILT_ENB" := "PDO".TCH_TILT_ENB XOR "IDO".TCH_TILT_ENB;
           "HDO_GTE_V_LFT_ENB" := "PDO".GTE_V_LFT_ENB XOR "IDO".GTE_V_LFT_ENB;
           "HDO_GTE_V_SW_ENB" := "PDO".GTE_V_SW_ENB XOR "IDO".GTE_V_SW_ENB;
           "HDO_BEL_LFT_ENB" := "PDO".BEL_LFT_ENB XOR "IDO".BEL_LFT_ENB;
           "HDO_HOR_OPP_K9" := "PDO".HOR_OPP_K9 XOR "IDO".HOR_OPP_K9;
           "HDO_LMP_RD_K9" := "PDO".LMP_RD_K9 XOR "IDO".LMP_RD_K9;
           "HDO_LMP_YE_K9" := "PDO".LMP_YE_K9 XOR "IDO".LMP_YE_K9;
           "HDO_LMP_GN_K9" := "PDO".LMP_GN_K9 XOR "IDO".LMP_GN_K9;
           "HDO_LMP_BU_K9" := "PDO".LMP_BU_K9 XOR "IDO".LMP_BU_K9;
       END_IF;
   END_IF;
END_FUNCTION_BLOCK

FUNCTION_BLOCK "PM_AI"   // FB19, SCL
{ S7_Optimized_Access := 'FALSE' }
VERSION : 0.0
// --------------------------------------------------------------------------------
//     program:         PM_AI
//     description :    automatically generated PM_AI
//     name:            hp
//     date        :    03.02.2021
// 
//     revision:
//     name:
//     Date:
//                     (c)CGS
//     --------------------------------------------------------------------------------
   VAR
      y : Bool;
      count : Int := 8;
   END_VAR
   VAR_TEMP
      x : Bool;
   END_VAR
BEGIN


   IF "SY".SIM_ON AND NOT "SY".SRM_ON THEN

       "PAI".TRV_ACT_POS := "SAI".TRV_ACT_POS;
       "PAI".TRV_ACT_POS_1 := "SAI".TRV_ACT_POS_1;
       "PAI".TRV_PRS_FIL_1 := "SAI".TRV_PRS_FIL_1;
       "PAI".TRV_PRS_FIL_2 := "SAI".TRV_PRS_FIL_2;
       "PAI".PYR_ACT_HTR_1_TMP := "SAI".PYR_ACT_HTR_1_TMP;
       "PAI".ACT_PRS_AR_VSL := "SAI".ACT_PRS_AR_VSL;
       "PAI".PYR_ACT_MELT_TMP := "SAI".PYR_ACT_MELT_TMP;
       "PAI".GCH_PCR_ACT_PRS := "SAI".GCH_PCR_ACT_PRS;
       "PAI".FCH_PCR_ACT_PRS := "SAI".FCH_PCR_ACT_PRS;
       "PAI".FCH_BAR_ACT_PRS_100 := "SAI".FCH_BAR_ACT_PRS_100;
       "PAI".ACC_WTR_TMP := "SAI".ACC_WTR_TMP;
       "PAI".ACC_WTR_PRS_IN := "SAI".ACC_WTR_PRS_IN;
       "PAI".ACC_WTR_FLW_OUT := "SAI".ACC_WTR_FLW_OUT;
       "PAI".ACC_WTR_FLW_IN := "SAI".ACC_WTR_FLW_IN;
       "PAI".ACC_WTR_SPL_PRS := "SAI".ACC_WTR_SPL_PRS;
       "PAI".ACC_SPARE_810 := "SAI".ACC_SPARE_810;
   ELSE

       "PAI".TRV_ACT_POS := "PM_AI_CONVERT" (CHANNEL := "HAI".TRV_ACT_POS, CONVERT_PAR:="CAI".CONFIG_DATA[1]);
       "PAI".TRV_ACT_POS_1 := "PM_AI_CONVERT" (CHANNEL := "HAI".TRV_ACT_POS_1, CONVERT_PAR:="CAI".CONFIG_DATA[2]);
       "PAI".TRV_PRS_FIL_1 := "PM_AI_CONVERT" (CHANNEL := "HAI".TRV_PRS_FIL_1, CONVERT_PAR:="CAI".CONFIG_DATA[3]);
       "PAI".TRV_PRS_FIL_2 := "PM_AI_CONVERT" (CHANNEL := "HAI".TRV_PRS_FIL_2, CONVERT_PAR:="CAI".CONFIG_DATA[4]);
       "PAI".PYR_ACT_HTR_1_TMP := "PM_AI_CONVERT" (CHANNEL := "HAI".PYR_ACT_HTR_1_TMP, CONVERT_PAR:="CAI".CONFIG_DATA[5]);
       "PAI".ACT_PRS_AR_VSL := "PM_AI_CONVERT" (CHANNEL := "HAI".ACT_PRS_AR_VSL, CONVERT_PAR:="CAI".CONFIG_DATA[6]);
       "PAI".PYR_ACT_MELT_TMP := "PM_AI_CONVERT" (CHANNEL := "HAI".PYR_ACT_MELT_TMP, CONVERT_PAR:="CAI".CONFIG_DATA[7]);
       "PAI".GCH_PCR_ACT_PRS := "PM_AI_CONVERT" (CHANNEL := "HAI".GCH_PCR_ACT_PRS, CONVERT_PAR:="CAI".CONFIG_DATA[8]);
       "PAI".FCH_PCR_ACT_PRS := "PM_AI_CONVERT" (CHANNEL := "HAI".FCH_PCR_ACT_PRS, CONVERT_PAR:="CAI".CONFIG_DATA[9]);
       "PAI".FCH_BAR_ACT_PRS_100 := "PM_AI_CONVERT" (CHANNEL := "HAI".FCH_BAR_ACT_PRS_100, CONVERT_PAR:="CAI".CONFIG_DATA[10]);
       "PAI".ACC_WTR_TMP := "PM_AI_CONVERT" (CHANNEL := "HAI".ACC_WTR_TMP, CONVERT_PAR:="CAI".CONFIG_DATA[11]);
       "PAI".ACC_WTR_PRS_IN := "PM_AI_CONVERT" (CHANNEL := "HAI".ACC_WTR_PRS_IN, CONVERT_PAR:="CAI".CONFIG_DATA[12]);
       "PAI".ACC_WTR_FLW_OUT := "PM_AI_CONVERT" (CHANNEL := "HAI".ACC_WTR_FLW_OUT, CONVERT_PAR:="CAI".CONFIG_DATA[13]);
       "PAI".ACC_WTR_FLW_IN := "PM_AI_CONVERT" (CHANNEL := "HAI".ACC_WTR_FLW_IN, CONVERT_PAR:="CAI".CONFIG_DATA[14]);
       "PAI".ACC_WTR_SPL_PRS := "PM_AI_CONVERT" (CHANNEL := "HAI".ACC_WTR_SPL_PRS, CONVERT_PAR:="CAI".CONFIG_DATA[15]);
       "PAI".ACC_SPARE_810 := "PM_AI_CONVERT" (CHANNEL := "HAI".ACC_SPARE_810, CONVERT_PAR:="CAI".CONFIG_DATA[16]);
   END_IF;
END_FUNCTION_BLOCK

FUNCTION_BLOCK "PM_AO"   // FB20, SCL
{ S7_Optimized_Access := 'FALSE' }
VERSION : 0.0
// --------------------------------------------------------------------------------
//     program:         PM_AO
//     description :    automatically generated PM_AO
//     name:            hp
//     date        :    03.02.2021
// 
//     revision:
//     name:
//     Date:
//                     (c)CGS
//     --------------------------------------------------------------------------------
   VAR
      y : Bool;
      count : Int := 8;
   END_VAR
   VAR_TEMP
      x : Bool;
   END_VAR
BEGIN


   IF "SY".SRM_ON THEN

       "HAO".TRV_SET_POS := "PM_AO_CONVERT"(OUTVALUE := "SAO".TRV_SET_POS, CONVERT_PAR := "CAO".CONFIG_DATA[1]);
       "HAO".TRV_SET_POS_1 := "PM_AO_CONVERT"(OUTVALUE := "SAO".TRV_SET_POS_1, CONVERT_PAR := "CAO".CONFIG_DATA[2]);
   ELSE
       IF NOT "SY".SIM_ON THEN

           "HAO".TRV_SET_POS := "PM_AO_CONVERT"(OUTVALUE := "PAO".TRV_SET_POS, CONVERT_PAR := "CAO".CONFIG_DATA[1]);
           "HAO".TRV_SET_POS_1 := "PM_AO_CONVERT"(OUTVALUE := "PAO".TRV_SET_POS_1, CONVERT_PAR := "CAO".CONFIG_DATA[2]);
       END_IF;
   END_IF;
END_FUNCTION_BLOCK

FUNCTION_BLOCK "PM_GET_WGT_XT_CLP"   // FB29, SCL
{ S7_Optimized_Access := 'FALSE' }
VERSION : 0.0
// --------------------------------------------------------------------------------
//     program     :    PM_GET_WGT_XT_CLP
//     description :    read load cell data and convert in weight unit   
//     name        :    lv
//     date        :    21.09.2016
// 
//     revision    :    
//     name        :
//     date        :    
//                     (c)CGS
//     --------------------------------------------------------------------------------
   VAR
      i : Int;
      bdg_vlt_clp_wgt : Real;   // bridge voltage load cell
      ref_vlt_clp_wgt : Real;   // reference voltage load cell
      start_si_lvl : Real;
      mess_si_lvl : Real;
      hop_cone : Real;
      hop_cute : Real;
      hop_cyl_start : Real;
      hop_cyl_mess : Real;
      hop_sum : Real;
      hop_mess : Real;
      tar_xt_clp_wgt : Bool;
      fl_tar_xt_clp_wgt : Bool;
   END_VAR
   VAR_TEMP
      Kl3351_1_IN : Struct
         D1_0 : Byte;   // High byte channel 1
         D0_0 : Byte;   // Low byte channel 1
         D1_1 : Byte;   // High byte channel 2
         D0_1 : Byte;   // Low byte channel 2
      END_STRUCT;
      Kl3351_1_OUT : Struct
         D1_0 : Byte;   // High byte channel 1
         D0_0 : Byte;   // Low byte channel 1
         D1_1 : Byte;   // High byte channel 2
         D0_1 : Byte;   // Low byte channel 2
      END_STRUCT;
      Dprd_RetVal_1 : Int;
      data_int : Int;
      data_word : Word;
      ctrl_byte : Byte;
      lb_data_word : Byte;
      hb_data_word : Byte;
   END_VAR
   VAR CONSTANT
      bdg_vlt_sca_fct : Real := 5.0E-07;   // bridge voltage scaling factor (500nV/digit) siehe Beckhoff Doku
      ref_vlt_sca_fct : Real := 0.0005;   // reference voltage scaling factor (500yV/digit) siehe Beckhoff Doku
      rtd_val_clp_wgt_cell : Real := 2.0E-05;   // 2 mV/V rated characteristic value crystal weight load cell
   END_VAR
BEGIN

       //---------------------------
       //read out process data feeder load cell
       //----------------------------------------------
       #Dprd_RetVal_1         := DPRD_DAT(LADDR :=  16#610,            //addr: 1552
                                           RECORD =>  #Kl3351_1_IN);
       //channel one
       //-----------
       //sta_byte_1          :=  Kl3351_1_IN.ST_0;  
       #lb_data_word        :=  #Kl3351_1_IN.D0_0;
       #hb_data_word        :=  #Kl3351_1_IN.D1_0;

       #data_word           :=  SHL(IN:=BYTE_TO_WORD(#hb_data_word), N:=8) OR BYTE_TO_WORD(#lb_data_word);
       #data_int            :=  WORD_TO_INT(#data_word);

       #bdg_vlt_clp_wgt          := (INT_TO_REAL(#data_int)) * #bdg_vlt_sca_fct;

       //channel two
       //-----------
       //sta_byte_2          :=  Kl3351_1_IN.ST_1;  
       #lb_data_word        :=  #Kl3351_1_IN.D0_1;
       #hb_data_word        :=  #Kl3351_1_IN.D1_1;

       #data_word           :=  SHL(IN:=BYTE_TO_WORD(#hb_data_word), N:=8) OR BYTE_TO_WORD(#lb_data_word);
       #data_int            :=  WORD_TO_INT(#data_word);

       #ref_vlt_clp_wgt     := (INT_TO_REAL(#data_int)) * #ref_vlt_sca_fct;


       //calculation of feeder cute weight in g
       //----------------------------------
       IF NOT "SY".SIM_ON    THEN                //simulation mode disabled?
           IF (#ref_vlt_clp_wgt > 0.0)   THEN 
               "AV".XT_HDL_CLP_WGT  := ((#bdg_vlt_clp_wgt / #ref_vlt_clp_wgt) * (10.0 / #rtd_val_clp_wgt_cell)) 
                                         * "CNF".XT_CLP_LDC_CAL;

           END_IF;
       END_IF;

      IF "PDI".LS_XT_CLP_CON THEN               // create auto calibration bit
         IF ("DIS".ACT_POS_XT_HDL_LFT>400.0) AND NOT "LT".XT_HDL_LFT_UP AND NOT "LT".XT_HDL_LFT_DN AND NOT #fl_tar_xt_clp_wgt THEN 
            #tar_xt_clp_wgt    := True;
            #fl_tar_xt_clp_wgt := True;
         END_IF;
      ELSE
         #tar_xt_clp_wgt    := false;
         #fl_tar_xt_clp_wgt := false;
      END_IF;        

       //set display variable
       //--------------------
       IF "PDI".LS_XT_CLP_CON OR "SysLog1" THEN
           "DIS".XT_HDL_CLP_WGT      :=  "AV".XT_HDL_CLP_WGT;   
           "DIS".XT_HDL_CLP_WGT_TAR  :=  "AV".XT_HDL_CLP_WGT - "AV".XT_HDL_CLP_TAR_WGT;
           IF "CNF".XT_CLP_LDC_CAL= 0.0 THEN
              "CNF".XT_CLP_LDC_CAL := 1.0;
           END_IF;
           IF ("KYD".XT_CLP_WGT_TAR) OR #tar_xt_clp_wgt THEN
               "AV".XT_HDL_CLP_TAR_WGT := "AV".XT_HDL_CLP_WGT;
               #tar_xt_clp_wgt := false;
           END_IF;     
       ELSE
           "DIS".XT_HDL_CLP_WGT      :=  0.0;   
           "DIS".XT_HDL_CLP_WGT_TAR  :=  0.0;
           "AV".XT_HDL_CLP_WGT       :=  0.0;   
           "AV".XT_HDL_CLP_TAR_WGT   :=  0.0;
       END_IF;
END_FUNCTION_BLOCK

FUNCTION_BLOCK "PM_TLU_PWR_SPL"   // FB33, SCL
{ S7_Optimized_Access := 'FALSE' }
VERSION : 0.0
// --------------------------------------------------------------------------------
//     program     :   PM_TLU_PWR_SPL  
//     description :   data transfer from and to TLU power supply profibus module
//     name        :   G. Eibelsh鋟ser  
//     date        :   16.04.2012
// 
//     revision    :
//     name        :
//     DATE        :    
//                     (c) PVATepla AG
//     --------------------------------------------------------------------------------
   VAR_INPUT
      htr_enb : Bool;   // heater enable
      htr_rst : Bool;   // heater reset
      fst_byte_offs : Int;   // first record byte in DB PM_TLU_PWR_SPL_DATA_BUF
      dp_adress : Word;   // address to read/write data from/to (DP Adress ID LADDR)
      set_htr_pwr : Real;
      htr_pwr_rng : Real;
      htr_cur_rng : Real;
      htr_vlt_rng : Real;
   END_VAR
   VAR_OUTPUT
      sta_htr_on : Bool;
      sta_error : Bool;
      sta_warn : Bool;
      sta_pi_mode : Bool;
      sta_pu_mode : Bool;
      sta_i_mode : Bool;
      sta_u_mode : Bool;
      sta_saved : Bool;
      flt_i_pri : Bool;
      flt_i_max : Bool;
      flt_u_max : Bool;
      flt_wire : Bool;
      flt_flash : Bool;
      flt_trafo : Bool;
      flt_data_flow : Bool;
      flt_data_com : Bool;
      flt_data : Bool;
      flt_tast : Bool;
      flt_ua_max : Bool;
      flt_u_min : Bool;
      flt_temp : Bool;
      flt_sense : Bool;
      flt_igbt : Bool;
      flt_dioden : Bool;
      flt_3 : Bool;
      flt_shunt : Bool;
      flt_board : Bool;
      flt_6 : Bool;
      flt_soft : Bool;
      flt_timeout : Bool;
      flt_short : Bool;
      act_htr_cur : Real;
      act_htr_vlt : Real;
      act_htr_pwr : Real;
   END_VAR
   VAR
      htr_word_sta_1 : Word;
      htr_word_flt_1 : Word;
      htr_word_flt_2 : Word;
      htr_word_flt_mem_1 : Word;
      htr_word_flt_mem_2 : Word;
      htr_word_cur_n : Word;
      htr_word_vlt_n : Word;
      htr_word_pwr_n : Word;
      htr_word_sta_2 : Word;
      htr_word_enrj_1 : Word;
      htr_word_enrj_2 : Word;
      htr_word_enrj_3 : Word;
      htr_word_pls : Word;
      htr_word_presc : Word;
      htr_word_firm : Word;
   END_VAR
   VAR_TEMP
      Buffer : "UDT_ANY_POINTER";
      Temp_Any_Pointer AT Buffer : ANY;
      RetVal : Int;   // Return Value of SFC 14/15
      DB_Byte_Adr : Int;   // start address in DB for reading/writing
      ctrl_low_byte : Byte;
      ctrl_high_byte : Byte;
      ctrl_word : Word;
      set_pwr_word : Word;
      set_cur_word : Word;
      set_vlt_word : Word;
      htr_word_cur : Word;
      htr_word_vlt : Word;
      htr_word_pwr : Word;
      set_pwr : Real;
      set_cur : Real;
      set_vlt : Real;
   END_VAR
   VAR CONSTANT
      DB_Number : Int := 127;   // number of buffer data block containing data of SFC 14/15
      Byte_Count : Int := 6;   // number of bytes to read/write consistently
      res : Int := 25000;   // resolution of TLU data
   END_VAR
BEGIN

       //preset values for 10 Byte Buffer for ANY_Pointer 
       //------------------------------------------------
       #Buffer.Syntax_Id := B#16#10;    // buffer length - MUST always be 16#10! (S7 needs 10 bytes to save the data of...
                                       // ...parameter of type 'ANY')                                                
       #Buffer.DataType := B#16#02;     // code f黵 data type 'BYTE'

       (************************************************************************************************************* 
          code for data types:
          --------------------
           b#16#00 = NIL,      b#16#01 = BOOL,     b#16#02 = BYTE,     b#16#03 = CHAR,     b#16#04 = WORD, b#16#05 = INT, 
           b#16#06 = DWORD,    b#16#07 = DINT,     b#16#08 = REAL,     b#16#09 = DATE,     b#16#0A = TIME_OF_DAY (TOD), 
           b#16#0B = TIME,     b#16#0C = S5TIME,   b#16#0E = DATE_AND_TIME (DT),           b#16#13 = STRING            
       **************************************************************************************************************) 

       #Buffer.Count        := INT_TO_WORD(32);          // number of bytes to read
       #Buffer.DB_Number    := INT_TO_WORD(#DB_Number);  
       (********************************************************************************** 
          code for memory area (=> highest byte of Buffer.Byte_Pointer)
          --------------------
           b#16#81 = E,    b#16#82 = A,    b#16#83 = M,    b#16#84 = DB,   b#16#85 = DI,
           b#16#86 = L,    b#16#87 = V
       ***********************************************************************************)
       //read the first Byte Block data from Plating profibus module Byte 0..31
       //----------------------------------
       #Buffer.Byte_Pointer := DW#16#8400_0000;                             // Null Pointer to global data DBX0.0 (code for memory data)
       #DB_Byte_Adr := #fst_byte_offs;                                       //set start byte address in DB PM_TLU_PWR_SPL_DATA_BUF for reading
       #Buffer.Byte_Pointer := #Buffer.Byte_Pointer OR (SHL(IN:=WORD_TO_DWORD(INT_TO_WORD(#DB_Byte_Adr)),N:=3));  // bits 0..2 of Byte_Pointer contain bit-add         
       #RetVal := DPRD_DAT(LADDR:= #dp_adress, RECORD=>#Temp_Any_Pointer);    // read values from periphery
       //---------------------------------------------------------------------------------------------------------------------

       //read the second Byte Block data from Plating profibus module 32..35
       #Buffer.Count        := INT_TO_WORD(4);          // number of bytes to read
       #Buffer.DB_Number    := INT_TO_WORD(#DB_Number);  

       (********************************************************************************** 
          code for memory area (=> highest byte of Buffer.Byte_Pointer)
          --------------------
           b#16#81 = E,    b#16#82 = A,    b#16#83 = M,    b#16#84 = DB,   b#16#85 = DI,
           b#16#86 = L,    b#16#87 = V
       ***********************************************************************************) 
       //----------------------------------
       #Buffer.Byte_Pointer := DW#16#8400_0000;                             // Null Pointer to global data DBX0.0 (code for memory data)
       #DB_Byte_Adr := #fst_byte_offs+32;                                       //set start byte address in DB PM_TLU_PWR_SPL_DATA_BUF for reading
       #Buffer.Byte_Pointer := #Buffer.Byte_Pointer OR (SHL(IN:=WORD_TO_DWORD(INT_TO_WORD(#DB_Byte_Adr)),N:=3));  // bits 0..2 of Byte_Pointer contain bit-add         
       #RetVal := DPRD_DAT(LADDR:= #dp_adress, RECORD=>#Temp_Any_Pointer);    // read values from periphery

       //read status byte and data word from input buffer
       //------------------------------------------------
       #htr_word_cur        :=  BYTE_TO_WORD(%DB127.DB(#fst_byte_offs + 0)) OR
                               SHL(IN:=BYTE_TO_WORD(%DB127.DB(#fst_byte_offs + 1)), N:=8);

       #htr_word_vlt        :=  BYTE_TO_WORD(%DB127.DB(#fst_byte_offs + 2)) OR
                               SHL(IN:=BYTE_TO_WORD(%DB127.DB(#fst_byte_offs + 3)), N:=8);

       #htr_word_sta_1      :=  BYTE_TO_WORD(%DB127.DB(#fst_byte_offs + 4)) OR
                               SHL(IN:=BYTE_TO_WORD(%DB127.DB(#fst_byte_offs + 5)), N:=8);

       #htr_word_pwr        :=  BYTE_TO_WORD(%DB127.DB(#fst_byte_offs + 6)) OR
                               SHL(IN:=BYTE_TO_WORD(%DB127.DB(#fst_byte_offs + 7)), N:=8);

       #htr_word_flt_mem_1  :=  BYTE_TO_WORD(%DB127.DB(#fst_byte_offs + 8)) OR
                               SHL(IN:=BYTE_TO_WORD(%DB127.DB(#fst_byte_offs + 9)), N:=8);

       #htr_word_flt_mem_2  :=  BYTE_TO_WORD(%DB127.DB(#fst_byte_offs + 10)) OR
                               SHL(IN:=BYTE_TO_WORD(%DB127.DB(#fst_byte_offs + 11)), N:=8);

       #htr_word_flt_1      :=  BYTE_TO_WORD(%DB127.DB(#fst_byte_offs + 12)) OR
                               SHL(IN:=BYTE_TO_WORD(%DB127.DB(#fst_byte_offs + 13)), N:=8);

       #htr_word_flt_2      :=  BYTE_TO_WORD(%DB127.DB(#fst_byte_offs + 14)) OR
                               SHL(IN:=BYTE_TO_WORD(%DB127.DB(#fst_byte_offs + 15)), N:=8);

       #htr_word_cur_n      :=  BYTE_TO_WORD(%DB127.DB(#fst_byte_offs + 16)) OR
                               SHL(IN:=BYTE_TO_WORD(%DB127.DB(#fst_byte_offs + 17)), N:=8);

       #htr_word_vlt_n      :=  BYTE_TO_WORD(%DB127.DB(#fst_byte_offs + 18)) OR
                               SHL(IN:=BYTE_TO_WORD(%DB127.DB(#fst_byte_offs + 19)), N:=8);

       #htr_word_pwr_n      :=  BYTE_TO_WORD(%DB127.DB(#fst_byte_offs + 20)) OR
                               SHL(IN:=BYTE_TO_WORD(%DB127.DB(#fst_byte_offs + 21)), N:=8);

       #htr_word_sta_2      :=  BYTE_TO_WORD(%DB127.DB(#fst_byte_offs + 22)) OR
                               SHL(IN:=BYTE_TO_WORD(%DB127.DB(#fst_byte_offs + 23)), N:=8);

       #htr_word_enrj_1     :=  BYTE_TO_WORD(%DB127.DB(#fst_byte_offs + 24)) OR
                               SHL(IN:=BYTE_TO_WORD(%DB127.DB(#fst_byte_offs + 25)), N:=8);

       #htr_word_enrj_2     :=  BYTE_TO_WORD(%DB127.DB(#fst_byte_offs + 26)) OR
                               SHL(IN:=BYTE_TO_WORD(%DB127.DB(#fst_byte_offs + 27)), N:=8);

       #htr_word_enrj_3     :=  BYTE_TO_WORD(%DB127.DB(#fst_byte_offs + 28)) OR
                               SHL(IN:=BYTE_TO_WORD(%DB127.DB(#fst_byte_offs + 29)), N:=8);

       #htr_word_pls        :=  BYTE_TO_WORD(%DB127.DB(#fst_byte_offs + 30)) OR
                               SHL(IN:=BYTE_TO_WORD(%DB127.DB(#fst_byte_offs + 31)), N:=8);

       #htr_word_presc      :=  BYTE_TO_WORD(%DB127.DB(#fst_byte_offs + 32)) OR
                               SHL(IN:=BYTE_TO_WORD(%DB127.DB(#fst_byte_offs + 33)), N:=8);

       #htr_word_firm       :=  BYTE_TO_WORD(%DB127.DB(#fst_byte_offs + 34)) OR
                               SHL(IN:=BYTE_TO_WORD(%DB127.DB(#fst_byte_offs + 35)), N:=8);


       //scale output variables
       //----------------------
       #act_htr_cur :=  DINT_TO_REAL(WORD_TO_DINT(#htr_word_cur)) / #res * #htr_cur_rng; 
       #act_htr_pwr :=  DINT_TO_REAL(WORD_TO_DINT(#htr_word_pwr)) / #res * #htr_pwr_rng;
       #act_htr_vlt :=  DINT_TO_REAL(WORD_TO_DINT(#htr_word_vlt)) / #res * #htr_vlt_rng;

       //evaluate status bits
       //--------------------
       //Betrieb 
       //-------
       IF ((#htr_word_sta_1 AND 2#0000_0001) = 2#0000_0001) THEN
           #sta_htr_on  := true;
       ELSE
           #sta_htr_on  := false;
       END_IF;  

       //Fehler 
       //------
       IF ((#htr_word_sta_1 AND 2#0000_0010) = 2#0000_0010) THEN
           #sta_error  := true;
       ELSE
           #sta_error  := false;
       END_IF;

       //Warnung 
       //-------
       IF ((#htr_word_sta_1 AND 2#0000_0100) = 2#0000_0100) THEN
           #sta_warn  := true;
       ELSE
           #sta_warn  := false;
       END_IF;

       //P-I Modus 
       //---------
       IF ((#htr_word_sta_1 AND 2#0000_1000) = 2#0000_1000) THEN
           #sta_pi_mode  := true;
       ELSE
           #sta_pi_mode  := false;
       END_IF;

       //P-U Modus
       //--------- 
       IF ((#htr_word_sta_1 AND 2#0001_0000) = 2#0001_0000) THEN
           #sta_pu_mode  := true;
       ELSE
           #sta_pu_mode  := false;
       END_IF;

       //I Modus 
       //-------
       IF ((#htr_word_sta_1 AND 2#0010_0000) = 2#0010_0000) THEN
            #sta_i_mode  := true;
       ELSE
            #sta_i_mode  := false;
       END_IF;

       //U Modus
       //------- 
       IF ((#htr_word_sta_1 AND 2#0100_0000) = 2#0100_0000) THEN
           #sta_u_mode   := true;
       ELSE
           #sta_u_mode   := false;
       END_IF;

       //Speichern erfolgt 
       //-----------------
       IF ((#htr_word_sta_1 AND 2#1000_0000) = 2#1000_0000) THEN
           #sta_saved   := true;
       ELSE
           #sta_saved   := false;
       END_IF;

       //evaluate fault bits
       //-------------------
       // 躡erstrom Stromwandler ? - Abschaltung
       IF ((#htr_word_flt_1 AND 2#0000_0000_0000_0001) = 2#0000_0000_0000_0001) THEN
           #flt_i_pri  := true;
       ELSE
           #flt_i_pri  := false;
       END_IF;

       // 躡erstrom FPGA ? - Abschaltung
       IF ((#htr_word_flt_1 AND 2#0000_0000_0000_0010) = 2#0000_0000_0000_0010) THEN
           #flt_i_max  := true;
       ELSE
           #flt_i_max  := false;
       END_IF;

       // 躡erspannung FPGA ? - Abschaltung nach 3s
       IF ((#htr_word_flt_1 AND 2#0000_0000_0000_0100) = 2#0000_0000_0000_0100) THEN
           #flt_u_max  := true;
       ELSE
           #flt_u_max  := false;
       END_IF;

       // Kabelfehler ? - Warnung
       IF ((#htr_word_flt_1 AND 2#0000_0000_0010_0000) = 2#0000_0000_0010_0000) THEN
           #flt_wire  := true;
       ELSE
           #flt_wire  := false;
       END_IF;

       // Datenflashfehler ? - Abschaltung
       IF ((#htr_word_flt_1 AND 2#0000_0000_0100_0000) = 2#0000_0000_0100_0000) THEN
           #flt_flash  := true;
       ELSE
           #flt_flash  := false;
       END_IF;

       // Trafo 黚erhitzt ? - Abschaltung
       IF ((#htr_word_flt_1 AND 2#0000_0000_1000_0000) = 2#0000_0000_1000_0000) THEN
           #flt_trafo  := true;
       ELSE
           #flt_trafo  := false;
       END_IF;

       // kein Datenfluss / fehlerhafte Daten ? - Abschaltung nach 3s
       IF ((#htr_word_flt_1 AND 2#0000_0001_0000_0000) = 2#0000_0001_0000_0000) THEN
           #flt_data_flow  := true;
       ELSE
           #flt_data_flow  := false;
       END_IF;

       // keine Daten黚ernahme ? - Abschaltung
       IF ((#htr_word_flt_1 AND 2#0000_0010_0000_0000) = 2#0000_0010_0000_0000) THEN
           #flt_data_com   := true;
       ELSE
           #flt_data_com   := false;
       END_IF;

       // fehlerhafte Daten ? - Abschaltung
       IF ((#htr_word_flt_1 AND 2#0000_0100_0000_0000) = 2#0000_0100_0000_0000) THEN
           #flt_data   := true;
       ELSE
           #flt_data   := false;
       END_IF;

       // Tastverh鋖tnis im Anschlag ? - Meldung "Kein Betrieb"
       IF ((#htr_word_flt_1 AND 2#0001_0000_0000_0000) = 2#0001_0000_0000_0000) THEN
           #flt_tast   := true;
       ELSE
           #flt_tast   := false;
       END_IF;

       // Ausgangs黚erspannung (Software) ? - Warnung
       IF ((#htr_word_flt_2 AND 2#0000_0000_0000_0010) = 2#0000_0000_0000_0010) THEN
           #flt_ua_max   := true;
       ELSE
           #flt_ua_max   := false;
       END_IF;

       // Unterspannung (Software) ? - Abschaltung nach 3s
       IF ((#htr_word_flt_2 AND 2#0000_0000_0000_1000) = 2#0000_0000_0000_1000) THEN
           #flt_u_min   := true;
       ELSE
           #flt_u_min   := false;
       END_IF;    

       // Temperaturwarnung ? - Warnung
       IF ((#htr_word_flt_2 AND 2#0000_0000_0001_0000) = 2#0000_0000_0001_0000) THEN
           #flt_temp   := true;
       ELSE
           #flt_temp   := false;
       END_IF; 

       // Ua_sense - Ua_Klemme >= max ? - Warnung
       IF ((#htr_word_flt_2 AND 2#0000_0000_0010_0000) = 2#0000_0000_0010_0000) THEN
           #flt_sense  := true;
       ELSE
           #flt_sense  := false;
       END_IF;

       // Temperatursensor_1 IGBT ? - Abschaltung
       IF ((#htr_word_flt_2 AND 2#0000_0000_0100_0000) = 2#0000_0000_0100_0000) THEN
           #flt_igbt   := true;
       ELSE
           #flt_igbt   := false;
       END_IF; 

       // Temperatursensor_2 Dioden ? - Abschaltung
       IF ((#htr_word_flt_2 AND 2#0000_0000_1000_0000) = 2#0000_0000_1000_0000) THEN
           #flt_dioden   := true;
       ELSE
           #flt_dioden   := false;
       END_IF;

       // Temperatursensor_3 ? - Abschaltung
       IF ((#htr_word_flt_2 AND 2#0000_0001_0000_0000) = 2#0000_0001_0000_0000) THEN
           #flt_3   := true;
       ELSE
           #flt_3   := false;
       END_IF;

       // Temperatursensor_4 Wasser,Shunt ? - Abschaltung
       IF ((#htr_word_flt_2 AND 2#0000_0010_0000_0000) = 2#0000_0010_0000_0000) THEN
           #flt_shunt   := true;
       ELSE
           #flt_shunt   := false;
       END_IF;

       // Temperatursensor_5 Leiterkarte ? - Abschaltung
       IF ((#htr_word_flt_2 AND 2#0000_0100_0000_0000) = 2#0000_0100_0000_0000) THEN
           #flt_board   := true;
       ELSE
           #flt_board   := false;
       END_IF;

       // Temperatursensor_6 ? - Abschaltung
       IF ((#htr_word_flt_2 AND 2#0000_1000_0000_0000) = 2#0000_1000_0000_0000) THEN
           #flt_6   := true;
       ELSE
           #flt_6   := false;
       END_IF;

       // Softwarefehler ? - Abschaltung
       IF ((#htr_word_flt_2 AND 2#0001_0000_0000_0000) = 2#0001_0000_0000_0000) THEN
           #flt_soft   := true;
       ELSE
           #flt_soft   := false;
       END_IF;    

       // Softwarefehler Timeout ? - Abschaltung
       IF ((#htr_word_flt_2 AND 2#0010_0000_0000_0000) = 2#0010_0000_0000_0000) THEN
           #flt_timeout   := true;
       ELSE
           #flt_timeout   := false;
       END_IF;     

       // Kurzschluss ? - Abschaltung
       IF ((#htr_word_flt_2 AND 2#1000_0000_0000_0000) = 2#1000_0000_0000_0000) THEN
           #flt_short   := true;
       ELSE
           #flt_short   := false;
       END_IF;   

       //write data to power supply
       //---------------------------
       IF #htr_rst  THEN
           #ctrl_word   :=  #ctrl_word OR 2#0000_0000_0000_0010;     // reset
       ELSIF #htr_enb THEN                                  
           #ctrl_word   := 2#0000_0000_0000_0001;                   // Schalte Netzteil EIN
           #set_pwr     := #set_htr_pwr;                             // Sollwert Leistung
           #set_cur     := #htr_cur_rng;                             // Stromlimit
           #set_vlt     := #htr_vlt_rng;                             // Spannungslimit
       ELSE
           #ctrl_word   := 2#0000_0000_0000_0000;                   // Schalte Netzteil AUS
           #set_pwr     := 0.0;                                     // Sollwert Leistung
           #set_cur     := 0.0;                                     // Stromlimit
           #set_vlt     := 0.0;                                     // Spannungslimit
       END_IF;

       //split control word in low byte and high byte
       //--------------------------------------------
       #ctrl_low_byte   := WORD_TO_BYTE(#ctrl_word);
       #ctrl_high_byte  := WORD_TO_BYTE(SHR(IN:= (#ctrl_word),N:=8));

       //scale set point variables
       //-------------------------
       #set_pwr := #set_pwr / #htr_pwr_rng * #res;
       #set_cur := #set_cur / #htr_cur_rng * #res;
       #set_vlt := #set_vlt / #htr_vlt_rng * #res;

       //convert from real to word
       //-------------------------
       #set_pwr_word := DINT_TO_WORD(REAL_TO_DINT(#set_pwr));
       #set_cur_word := DINT_TO_WORD(REAL_TO_DINT(#set_cur));    
       #set_vlt_word := DINT_TO_WORD(REAL_TO_DINT(#set_vlt));

       //write control byte and data word to data buffer
       //-----------------------------------------------
       %DB127.DB(#fst_byte_offs + 36) := WORD_TO_BYTE(#set_cur_word);
       %DB127.DB(#fst_byte_offs + 37) := WORD_TO_BYTE(SHR(IN:= #set_cur_word ,N:=8));
       %DB127.DB(#fst_byte_offs + 38) := WORD_TO_BYTE(#set_vlt_word);
       %DB127.DB(#fst_byte_offs + 39) := WORD_TO_BYTE(SHR(IN:= #set_vlt_word ,N:=8));
       %DB127.DB(#fst_byte_offs + 40) := #ctrl_low_byte;
       %DB127.DB(#fst_byte_offs + 41) := #ctrl_high_byte;
       %DB127.DB(#fst_byte_offs + 42) := WORD_TO_BYTE(#set_pwr_word);
       %DB127.DB(#fst_byte_offs + 43) := WORD_TO_BYTE(SHR(IN:= #set_pwr_word ,N:=8));

       //write data to TLU Profibus module
       //---------------------------------
       #Buffer.Count        := INT_TO_WORD(16);             // number of bytes to write
       #Buffer.Byte_Pointer := DW#16#8400_0000;             //Null Pointer to global data DBX0.0 (code for memory data)
       #DB_Byte_Adr := (#fst_byte_offs + 36);                //set start byte address in DB PM_TLU_PWR_SPL_DATA_BUF for writing
       #Buffer.Byte_Pointer := #Buffer.Byte_Pointer OR (SHL(IN:=WORD_TO_DWORD(INT_TO_WORD(#DB_Byte_Adr)),N:=3));    
       #RetVal := DPWR_DAT(LADDR:= #dp_adress, RECORD:=#Temp_Any_Pointer);     // write data to periphery
END_FUNCTION_BLOCK

FUNCTION_BLOCK "PM_DRV_COMM_LZI550"   // FB34, SCL
{ S7_Optimized_Access := 'FALSE' }
VERSION : 0.0
// --------------------------------------------------------------------------------
//     program     :    FB_DRV_COMM_LZI950
//     description :    communication with Lenze i950 
//     
//     name        :    L. Ewert
//     date        :    28.08.2018
// 
//     revision    :
//     name        :
//     date        :    
//                     (c)PVATepla
//     --------------------------------------------------------------------------------
   VAR_INPUT
      Enable : Bool;   // Enable speed controll
      CW : Bool;   // Turn direction clock wise
      CCW : Bool;   // Turn direction counter clock wise
      Stopp : Bool;   // Ends CW / CCW
      Reset_error : Bool;   // Reset actual Error
      PM_ADR_A : Word;   // Periphery-Adress of the first output Word
      PM_ADR_E : Word;   // Periphery-Adress of the first input Word
      Speed_Hz : Real;   // Speed in Hz 50.00 Hz
   END_VAR
   VAR_OUTPUT
      Error : Bool;   // Error Bit
      Ready : Bool;   // Drive is ready for CW / CCW
      Speed_reached : Bool;   // Act_Speed = Set_Speed
      Running : Bool;   // Drive is running
      Error_code : DInt;   // Number of actual Error
      Act_Speed_Hz : Real;   // Actual Speed in Hz
   END_VAR
   VAR
      W_CTLW : Word;
      B_CTLW AT W_CTLW : Array[0..1] of Byte;
      W_STATW : Word;
      B_STATW AT W_STATW : Array[0..1] of Byte;
      DRV_DATA_i550 : "UDT_DRV_LENZE_i550";
      RD_DATA : Struct
         HI_BYTE : Byte;
         LO_BYTE : Byte;
      END_STRUCT;
      RD_DATA_W AT RD_DATA : Word;
      WR_DATA_W : Word;
      WR_DATA AT WR_DATA_W : Struct
         HI_BYTE : Byte;
         LO_BYTE : Byte;
      END_STRUCT;
   END_VAR
   VAR_TEMP
      temp_Word_rd : Word;
      temp_b_ctlw AT temp_Word_rd : Array[0..1] of Byte;
      temp_x_ctlw AT temp_Word_rd : Array[0..15] of Bool;
      temp_Word_wr : Word;
      temp_b_statw AT temp_Word_wr : Array[0..1] of Byte;
      temp_x_statw AT temp_Word_wr : Array[0..15] of Bool;
      Error_Write_Data : Int;
      Error_Read_Data : Int;
      ADR_TMP : Word;
   END_VAR
BEGIN


       (*Statuswort f黵 i550 von Lenze
           Bez.            BIT Nr.
           Betriebsbereit    0
           Spare             1
           Freigabe          2
           Drive Fault       3
           Spare             4
           Quickstop Active  5
           In Betrieb        6
           Ger鋞ewarnung     7
           Spare             8
           Spare             9
           In Velocity (Istgeschwindigkeit entspricht Sollgeschwindigkeit)    10
           Stromlimit err.   11
           Standstill        12
           Dreh. umkehr      13
           Brake Released    14
           STO Active        15
       *)
       (*Steuerwort f黵 i550 von Lenze
           Spare             0
           Reglersperre      1
           Stopp             2
           Quickstopp        3
           Fehler_reset      4
           DC_Bremse         5
           Run_Vorw鋜ts      6
           Run_R點kw鋜ts     7
           Drehrichtung_umk. 8
           NET_Sollw_vorg    9
           Spare             10
           Spare             11
           Spare             12
           Spare             13
           Spare             14
           Spare             15
       *)
       // W_CTLW is been set with the Byte Array B_CTLW

       // Swap the two Bytes of the Word because SCL will Set Bits in a Word from  LSB 8..15 0..7 MSB
       // Read Drive Data into Word
       #temp_b_ctlw[0]:= #B_CTLW[1];
       #temp_b_ctlw[1]:= #B_CTLW[0];

       #temp_x_ctlw[9]:= #Enable; // Set Bit 9 -> Enable Set Vel over NET
       #temp_x_ctlw[4]:= #Reset_error; // Set Bit 4 (Reset Error)
       IF #CW AND NOT #Stopp THEN
           #temp_x_ctlw[6]:= TRUE;      // Set Bit 6 (CW)
           #temp_x_ctlw[7]:= FALSE;     // Set Bit 7 back (CCW)
       ELSIF #CCW AND NOT #Stopp THEN
           #temp_x_ctlw[7]:= TRUE;      // Set Bit 7 (CCW)
           #temp_x_ctlw[6]:= FALSE;     // Set Bit 6 back (CW)        
       ELSE 
           #temp_x_ctlw[6]:= FALSE;     // Set Bit 6 back (CW)
           #temp_x_ctlw[7]:= FALSE;     // Set Bit 7 back (CCW)
       END_IF;

       #DRV_DATA_i550.Output.SET_Speed_Hz_0_1 := INT_TO_WORD(REAL_TO_INT(#Speed_Hz*100.0));    // Set Vel. in [Hz] 50.01 (SPS) -> 5001 (Drive) 

       // Swap the two Bytes of the Word because SCL will Set Bits in a Word from  LSB 8..15 0..7 MSB
       #B_CTLW[0]:=#temp_b_ctlw[1];
       #B_CTLW[1]:=#temp_b_ctlw[0];
       #DRV_DATA_i550.Output.CTRW:= #W_CTLW;
       // Write Data to Drive   
       #WR_DATA_W := #DRV_DATA_i550.Output.CTRW;    
       #Error_Write_Data:= DPWR_DAT ( LADDR:= #PM_ADR_A, 
                                    RECORD:= #WR_DATA);

       #WR_DATA_W := #DRV_DATA_i550.Output.SET_Speed_Hz_0_1; 
       #Error_Write_Data:= DPWR_DAT ( LADDR:= INT_TO_WORD(WORD_TO_INT(#PM_ADR_A)+2), 
                                    RECORD:= #WR_DATA);

       // End Set Values 


       //actual motor values
       //---------------------  
       // Read data from Drive
       #Error_Read_Data:= DPRD_DAT ( LADDR := #PM_ADR_E, 
                                    RECORD=> #RD_DATA);
       #DRV_DATA_i550.Input.STATW := #RD_DATA_W;

       #Error_Read_Data:= DPRD_DAT ( LADDR := INT_TO_WORD(WORD_TO_INT(#PM_ADR_E)+2), 
                                    RECORD=> #RD_DATA);
       #DRV_DATA_i550.Input.ACT_Speed_Hz_0_1 := #RD_DATA_W;

       #Error_Read_Data:= DPRD_DAT ( LADDR := INT_TO_WORD(WORD_TO_INT(#PM_ADR_E)+6), 
                                    RECORD=> #RD_DATA);
       #DRV_DATA_i550.Input.Error_code  := #RD_DATA_W;

       #W_STATW:= #DRV_DATA_i550.Input.STATW;                               
       #temp_b_statw[0]:= #B_STATW[1];
       #temp_b_statw[1]:= #B_STATW[0];     
       #Act_Speed_Hz:=  INT_TO_REAL(WORD_TO_INT(#DRV_DATA_i550.Input.ACT_Speed_Hz_0_1))/100.0; // Read Vel. in [Hz] 5001 (Drive) -> 50.01 (SPS)

       #Ready:= #temp_x_statw[3]; // Read Status Ready from Drive 
       #Running:= #temp_x_statw[6]; // Read Status Ready from Drive  
       #Speed_reached:= #temp_x_statw[10]; // Drive Set-Speed = Act-Speed
       //actual fault
       //---------------------
       #Error_code:= INT_TO_DINT(WORD_TO_INT(#DRV_DATA_i550.Input.Error_code));    // Fehlernummer Umrichter
       #Error:= #temp_x_statw[3]; // Fehlerbit Umrichter
END_FUNCTION_BLOCK

FUNCTION_BLOCK "PM_INJET_PWR_SPL"   // FB35, SCL
{ S7_Optimized_Access := 'FALSE' }
VERSION : 0.0
// --------------------------------------------------------------------------------
//     program     :    PM_INJET_PWR_SPL
//     description :    data transfer from and to Injet power supply
//                      
//  
//     name        :    John Wang
//     date        :    25.03.2020
// 
//     revision    :    
//     name        :    
//     date        :     
//      
//                     (c)PVATEPLA
//     --------------------------------------------------------------------------------
   VAR_INPUT
      htr_1_enb : Bool;   // heater 1 enable
      htr_2_enb : Bool;   // heater 1 enable
      set_htr_1_pwr : Real;   // set heater 1 power
      set_htr_2_pwr : Real;   // set heater 2 power
   END_VAR
   VAR_OUTPUT
      flt_pwr_spl_panel_comm : Bool;
      flt_pwr_spl_APF : Bool;
      flt_htr1_rct_tmp : Bool;
      flt_htr2_rct_tmp : Bool;
      htr_1_remote : Bool;
      comm_ok : Bool;
      htr_pwr_spl_cool_wtr_flt : Bool;
      htr_pwr_spl_cool_wtr_wrn : Bool;
      htr_1_flt_ctrl : Bool;
      htr_1_flt_comm : Bool;
      htr_1_flt_save : Bool;
      htr_1_flt_ac_pha : Bool;
      htr_1_flt_tmp : Bool;
      htr_1_flt_cur : Bool;
      htr_1_flt_cool_wtr : Bool;
      htr_1_flt_erd_plus : Bool;
      htr_1_flt_erd_min : Bool;
      htr_1_flt_term : Bool;
      htr_1_mod1_flt_syn_kab : Bool;
      htr_1_mod1_flt_sys_tmp : Bool;
      htr_1_mod1_flt_drv : Bool;
      htr_1_mod1_flt_cur : Bool;
      htr_1_mod1_flt_vlt : Bool;
      htr_1_mod1_flt_save : Bool;
      htr_1_mod1_flt_rect : Bool;
      htr_1_mod1_flt_tmp : Bool;
      htr_1_mod2_flt_syn_kab : Bool;
      htr_1_mod2_flt_sys_tmp : Bool;
      htr_1_mod2_flt_drv : Bool;
      htr_1_mod2_flt_cur : Bool;
      htr_1_mod2_flt_vlt : Bool;
      htr_1_mod2_flt_save : Bool;
      htr_1_mod2_flt_rect : Bool;
      htr_1_mod2_flt_tmp : Bool;
      htr_1_mod3_flt_syn_kab : Bool;
      htr_1_mod3_flt_sys_tmp : Bool;
      htr_1_mod3_flt_drv : Bool;
      htr_1_mod3_flt_cur : Bool;
      htr_1_mod3_flt_vlt : Bool;
      htr_1_mod3_flt_save : Bool;
      htr_1_mod3_flt_rect : Bool;
      htr_1_mod3_flt_tmp : Bool;
      htr_1_mod4_flt_syn_kab : Bool;
      htr_1_mod4_flt_sys_tmp : Bool;
      htr_1_mod4_flt_drv : Bool;
      htr_1_mod4_flt_cur : Bool;
      htr_1_mod4_flt_vlt : Bool;
      htr_1_mod4_flt_save : Bool;
      htr_1_mod4_flt_rect : Bool;
      htr_1_mod4_flt_tmp : Bool;
      htr_1_act_vlt : Real;
      htr_1_act_pwr : Real;
      htr_1_act_cur : Real;
      htr_1_act_resi : Real;
      htr_1_eth_vlt_plus : Real;
      htr_1_eth_vlt_minus : Real;
      htr_2_remote : Bool;
      htr_2_flt_ctrl : Bool;
      htr_2_flt_comm : Bool;
      htr_2_flt_save : Bool;
      htr_2_flt_ac_pha : Bool;
      htr_2_flt_tmp : Bool;
      htr_2_flt_cur : Bool;
      htr_2_flt_cool_wtr : Bool;
      htr_2_flt_erd_plus : Bool;
      htr_2_flt_erd_min : Bool;
      htr_2_flt_term : Bool;
      htr_2_mod1_flt_syn_kab : Bool;
      htr_2_mod1_flt_sys_tmp : Bool;
      htr_2_mod1_flt_drv : Bool;
      htr_2_mod1_flt_cur : Bool;
      htr_2_mod1_flt_vlt : Bool;
      htr_2_mod1_flt_save : Bool;
      htr_2_mod1_flt_rect : Bool;
      htr_2_mod1_flt_tmp : Bool;
      htr_2_mod2_flt_syn_kab : Bool;
      htr_2_mod2_flt_sys_tmp : Bool;
      htr_2_mod2_flt_drv : Bool;
      htr_2_mod2_flt_cur : Bool;
      htr_2_mod2_flt_vlt : Bool;
      htr_2_mod2_flt_save : Bool;
      htr_2_mod2_flt_rect : Bool;
      htr_2_mod2_flt_tmp : Bool;
      htr_2_mod3_flt_syn_kab : Bool;
      htr_2_mod3_flt_sys_tmp : Bool;
      htr_2_mod3_flt_drv : Bool;
      htr_2_mod3_flt_cur : Bool;
      htr_2_mod3_flt_vlt : Bool;
      htr_2_mod3_flt_save : Bool;
      htr_2_mod3_flt_rect : Bool;
      htr_2_mod3_flt_tmp : Bool;
      htr_2_act_vlt : Real;
      htr_2_act_pwr : Real;
      htr_2_act_cur : Real;
      htr_2_act_resi : Real;
      htr_2_eth_vlt_plus : Real;
      htr_2_eth_vlt_minus : Real;
   END_VAR
   VAR
      PWR_SPL_CTRL_W : Word;
      PWR_SPL_CTRL AT PWR_SPL_CTRL_W : Struct
         B00_HTR_1_ON : Bool;   // heater 1 power on
         B01_spare : Bool;
         B02_HTR_2_ON : Bool;   // heater 2 power on
         B03_spare : Bool;
         B04_spare : Bool;
         B05_spare : Bool;
         B06_spare : Bool;
         B07_spare : Bool;
         B10_spare : Bool;
         B11_spare : Bool;
         B12_spare : Bool;
         B13_spare : Bool;
         B14_spare : Bool;
         B15_spare : Bool;
         B16_spare : Bool;
         B17_spare : Bool;
      END_STRUCT;
      PWR_SPL_1_SET_PWR : Real;   // heater set power
      PWR_SPL_2_SET_PWR : Real;   // heater set power
      PWR_SPL_STAT_W : Word;
      PWR_SPL_STAT_B AT PWR_SPL_STAT_W : Struct
         PWR_SPL_STAT_L : Byte;
         PWR_SPL_STAT_H : Byte;
      END_STRUCT;
      PWR_SPL_STAT_BI AT PWR_SPL_STAT_W : Array[0..15] of Bool;
      PWR_SPL_STAT2_W : Word;
      PWR_SPL_STAT2_B AT PWR_SPL_STAT2_W : Struct
         PWR_SPL_STAT2_L : Byte;
         PWR_SPL_STAT2_H : Byte;
      END_STRUCT;
      PWR_SPL_STAT2_BI AT PWR_SPL_STAT2_W : Array[0..15] of Bool;
      PWR_SPL_STAT3_W : Word;
      PWR_SPL_STAT3_B AT PWR_SPL_STAT3_W : Struct
         PWR_SPL_STAT3_L : Byte;
         PWR_SPL_STAT3_H : Byte;
      END_STRUCT;
      PWR_SPL_STAT3_BI AT PWR_SPL_STAT3_W : Array[0..15] of Bool;
      PWR_SPL_STAT4_W : Word;
      PWR_SPL_STAT4_B AT PWR_SPL_STAT4_W : Struct
         PWR_SPL_STAT4_L : Byte;
         PWR_SPL_STAT4_H : Byte;
      END_STRUCT;
      PWR_SPL_STAT4_BI AT PWR_SPL_STAT4_W : Array[0..15] of Bool;
      PWR_SPL_STAT5_W : Word;
      PWR_SPL_STAT5_B AT PWR_SPL_STAT5_W : Struct
         PWR_SPL_STAT5_L : Byte;
         PWR_SPL_STAT5_H : Byte;
      END_STRUCT;
      PWR_SPL_STAT5_BI AT PWR_SPL_STAT5_W : Array[0..15] of Bool;
      PWR_SPL_STAT6_W : Word;
      PWR_SPL_STAT6_B AT PWR_SPL_STAT6_W : Struct
         PWR_SPL_STAT6_L : Byte;
         PWR_SPL_STAT6_H : Byte;
      END_STRUCT;
      PWR_SPL_STAT6_BI AT PWR_SPL_STAT6_W : Array[0..15] of Bool;
      PWR_SPL_STAT7_W : Word;
      PWR_SPL_STAT7_B AT PWR_SPL_STAT7_W : Struct
         PWR_SPL_STAT7_L : Byte;
         PWR_SPL_STAT7_H : Byte;
      END_STRUCT;
      PWR_SPL_STAT7_BI AT PWR_SPL_STAT7_W : Array[0..15] of Bool;
      PWR_SPL_1_ACT_VLT : Real;   // heater 1 act. voltage
      PWR_SPL_1_ACT_PWR : Real;   // heater 1 akt. power
      PWR_SPL_1_ACT_CUR : Real;   // heater 1 akt. current
      PWR_SPL_1_ACT_RESIS : Real;   // heater 1 akt. resistance
      PWR_SPL_1_BUS_PLUS : Real;   // heater 1 bus+
      PWR_SPL_1_BUS_MINUS : Real;   // heater 1 bus-
      PWR_SPL_2_ACT_VLT : Real;   // heater 2 act. voltage
      PWR_SPL_2_ACT_PWR : Real;   // heater 2 akt. power
      PWR_SPL_2_ACT_CUR : Real;   // heater 2 akt. current
      PWR_SPL_2_ACT_RESIS : Real;   // heater 2 akt. resistance
      PWR_SPL_2_BUS_PLUS : Real;   // heater 2 bus+
      PWR_SPL_2_BUS_MINUS : Real;   // heater 2 bus-
   END_VAR
BEGIN


   //--------------------------------------------
   //write a control word to Injet power supply

   "P_BM_PWR_SPL_CTRL":P    :=  WORD_TO_BYTE(SHR(IN :=#PWR_SPL_CTRL_W,N :=8));

   //--------------------------------------------
   //read status words from Injet power supply

   #PWR_SPL_STAT_W     :=  "P_BM_PWR_SPL_STAT":P;
   #PWR_SPL_STAT2_W     := "P_BM_PWR_SPL_STAT2":P; 
   #PWR_SPL_STAT3_W     := "P_BM_PWR_SPL_STAT3":P;
   #PWR_SPL_STAT4_W     := "P_BM_PWR_SPL_STAT4":P;
   #PWR_SPL_STAT5_W     := "P_BM_PWR_SPL_STAT5":P;
   #PWR_SPL_STAT6_W     := "P_BM_PWR_SPL_STAT6":P;
   #PWR_SPL_STAT7_W     := "P_BM_PWR_SPL_STAT7":P;

   #PWR_SPL_1_ACT_VLT   := "P_BM_PWR_SPL_1_ACT_VLT":P;
   #PWR_SPL_1_ACT_PWR   := "P_BM_PWR_SPL_1_ACT_PWR":P;
   #PWR_SPL_1_ACT_CUR   := "P_BM_PWR_SPL_1_ACT_CUR":P;
   #PWR_SPL_1_ACT_RESIS := "P_BM_PWR_SPL_1_ACT_RESIS":P;
   #PWR_SPL_1_BUS_PLUS  := "P_BM_PWR_SPL_1_BUS_PLUS":P;
   #PWR_SPL_1_BUS_MINUS := "P_BM_PWR_SPL_1_BUS_MINUS":P;

   #PWR_SPL_2_ACT_VLT   := "P_BM_PWR_SPL_2_ACT_VLT":P;
   #PWR_SPL_2_ACT_PWR   := "P_BM_PWR_SPL_2_ACT_PWR":P;
   #PWR_SPL_2_ACT_CUR   := "P_BM_PWR_SPL_2_ACT_CUR":P;
   #PWR_SPL_2_ACT_RESIS := "P_BM_PWR_SPL_2_ACT_RESIS":P;
   #PWR_SPL_2_BUS_PLUS  := "P_BM_PWR_SPL_2_BUS_PLUS":P;
   #PWR_SPL_2_BUS_MINUS := "P_BM_PWR_SPL_2_BUS_MINUS":P;

   #htr_1_act_vlt       := #PWR_SPL_1_ACT_VLT;
   #htr_1_act_pwr       := #PWR_SPL_1_ACT_PWR;
   #htr_1_act_resi      := #PWR_SPL_1_ACT_RESIS;
   #htr_1_act_cur       := #PWR_SPL_1_ACT_CUR;
   #htr_1_eth_vlt_plus  := #PWR_SPL_1_BUS_PLUS;
   #htr_1_eth_vlt_minus := #PWR_SPL_1_BUS_MINUS;

   #htr_2_act_vlt       := #PWR_SPL_2_ACT_VLT;
   #htr_2_act_pwr       := #PWR_SPL_2_ACT_PWR;
   #htr_2_act_cur       := #PWR_SPL_2_ACT_CUR;
   #htr_2_eth_vlt_plus  := #PWR_SPL_2_BUS_PLUS;
   #htr_2_eth_vlt_minus := #PWR_SPL_2_BUS_MINUS;       

   //--------------------------------------------
   //read bits from Injet power supply status words

   #htr_1_remote                :=     #PWR_SPL_STAT_BI[8];                     // heater 1 remote
   #htr_2_remote                :=     #PWR_SPL_STAT_BI[9];                     // heater 2 remote 
   #comm_ok                     :=     #PWR_SPL_STAT_BI[10];                    // communication is ok 

   #htr_pwr_spl_cool_wtr_flt    :=     #PWR_SPL_STAT2_BI[1];                    // cooling water fault
   #htr_pwr_spl_cool_wtr_wrn    :=     #PWR_SPL_STAT2_BI[2];                    // cooling water fault power off
   #flt_pwr_spl_APF             :=     #PWR_SPL_STAT2_BI[3];                    // APF fault
   #flt_htr1_rct_tmp            :=     #PWR_SPL_STAT2_BI[4];                    // heater 1 filter reactor temperature too high, more than 85癈
   #htr_1_flt_ctrl              :=     #PWR_SPL_STAT2_BI[5];                    // heater 1 controller fault
   #htr_2_flt_ctrl              :=     #PWR_SPL_STAT2_BI[6];                    // heater 2 controller fault 
   #htr_1_flt_comm              :=     #PWR_SPL_STAT2_BI[8];                    // heater 1 communication fault
   #htr_2_flt_comm              :=     #PWR_SPL_STAT2_BI[9];                    // heater 2 communication fault
   #flt_pwr_spl_panel_comm      :=     #PWR_SPL_STAT2_BI[10];                   // panel coomunication fault

   #htr_1_flt_save              :=     #PWR_SPL_STAT3_BI[0];                    // heater 1 save fault
   #htr_1_flt_ac_pha            :=     #PWR_SPL_STAT3_BI[1];                    // heater 1 AC phase
   #htr_1_flt_tmp               :=     #PWR_SPL_STAT3_BI[2];                    // heater 1 system temperature fault
   #htr_1_flt_cur               :=     #PWR_SPL_STAT3_BI[3];                    // heater 1 overcurrent 
   #htr_1_flt_cool_wtr          :=     #PWR_SPL_STAT3_BI[4];                    // heater 1 cooling water fault 
   #htr_1_flt_erd_plus          :=     #PWR_SPL_STAT3_BI[5];                    // heater 1 earthing plus fault  
   #htr_1_flt_erd_min           :=     #PWR_SPL_STAT3_BI[6];                    // heater 1 earthing minus fault 
   #htr_1_flt_term              :=     #PWR_SPL_STAT3_BI[7];                    // heater 1 terminal fault 


   // --------fault heater 1 modul 1

   #htr_1_mod1_flt_syn_kab      :=     #PWR_SPL_STAT3_BI[8];                     // synchronous cable fault
   #htr_1_mod1_flt_sys_tmp      :=     #PWR_SPL_STAT3_BI[9];                     // system temperature fault 
   #htr_1_mod1_flt_drv          :=     #PWR_SPL_STAT3_BI[10];                    // drive fault
   #htr_1_mod1_flt_cur          :=     #PWR_SPL_STAT3_BI[11];                    // overcurrent 
   #htr_1_mod1_flt_vlt          :=     #PWR_SPL_STAT3_BI[12];                    // voltage fault 
   #htr_1_mod1_flt_save         :=     #PWR_SPL_STAT3_BI[13];                    // save fault
   #htr_1_mod1_flt_rect         :=     #PWR_SPL_STAT3_BI[14];                    // rectification fault
   #htr_1_mod1_flt_tmp          :=     #PWR_SPL_STAT3_BI[15];                    // temperature fault 

   //---------fault heater 1 modul 2
   #htr_1_mod2_flt_syn_kab      :=     #PWR_SPL_STAT4_BI[0]; 
   #htr_1_mod2_flt_sys_tmp      :=     #PWR_SPL_STAT4_BI[1]; 
   #htr_1_mod2_flt_drv          :=     #PWR_SPL_STAT4_BI[2];
   #htr_1_mod2_flt_cur          :=     #PWR_SPL_STAT4_BI[3];
   #htr_1_mod2_flt_vlt          :=     #PWR_SPL_STAT4_BI[4];
   #htr_1_mod2_flt_save         :=     #PWR_SPL_STAT4_BI[5];
   #htr_1_mod2_flt_rect         :=     #PWR_SPL_STAT4_BI[6];
   #htr_1_mod2_flt_tmp          :=     #PWR_SPL_STAT4_BI[7];

   //---------fault heater 1 modul 3
   #htr_1_mod3_flt_syn_kab      :=     #PWR_SPL_STAT4_BI[8];
   #htr_1_mod3_flt_sys_tmp      :=     #PWR_SPL_STAT4_BI[9];
   #htr_1_mod3_flt_drv          :=     #PWR_SPL_STAT4_BI[10];
   #htr_1_mod3_flt_cur          :=     #PWR_SPL_STAT4_BI[11];
   #htr_1_mod3_flt_vlt          :=     #PWR_SPL_STAT4_BI[12];
   #htr_1_mod3_flt_save         :=     #PWR_SPL_STAT4_BI[13];
   #htr_1_mod3_flt_rect         :=     #PWR_SPL_STAT4_BI[14];
   #htr_1_mod3_flt_tmp          :=     #PWR_SPL_STAT4_BI[15];

   //---------fault heater 1 modul 4
   #htr_1_mod4_flt_syn_kab      :=     #PWR_SPL_STAT5_BI[0];
   #htr_1_mod4_flt_sys_tmp      :=     #PWR_SPL_STAT5_BI[1];
   #htr_1_mod4_flt_drv          :=     #PWR_SPL_STAT5_BI[2];
   #htr_1_mod4_flt_cur          :=     #PWR_SPL_STAT5_BI[3];
   #htr_1_mod4_flt_vlt          :=     #PWR_SPL_STAT5_BI[4];
   #htr_1_mod4_flt_save         :=     #PWR_SPL_STAT5_BI[5];
   #htr_1_mod4_flt_rect         :=     #PWR_SPL_STAT5_BI[6];
   #htr_1_mod4_flt_tmp          :=     #PWR_SPL_STAT5_BI[7];
   //---------------------------
   // fault heater 1 


   #htr_2_flt_save              :=     #PWR_SPL_STAT5_BI[8];                    // heater 2 save fault
   #htr_2_flt_ac_pha            :=     #PWR_SPL_STAT5_BI[9];                    // heater 2 AC phase
   #htr_2_flt_tmp               :=     #PWR_SPL_STAT5_BI[10];                   // heater 2 system temperature fault
   #htr_2_flt_cur               :=     #PWR_SPL_STAT5_BI[11];                   // heater 2 overcurrent 
   #htr_2_flt_cool_wtr          :=     #PWR_SPL_STAT5_BI[12];                   // heater 2 cooling water fault 
   #htr_2_flt_erd_plus          :=     #PWR_SPL_STAT5_BI[13];                   // heater 2 earthing plus fault  
   #htr_2_flt_erd_min           :=     #PWR_SPL_STAT5_BI[14];                   // heater 2 earthing minus fault 
   #htr_2_flt_term              :=     #PWR_SPL_STAT5_BI[15];                   // heater 2 terminal fault 

   //---------fault heater 2 modul 1
   #htr_2_mod1_flt_syn_kab      :=     #PWR_SPL_STAT6_BI[0];
   #htr_2_mod1_flt_sys_tmp      :=     #PWR_SPL_STAT6_BI[1];
   #htr_2_mod1_flt_drv          :=     #PWR_SPL_STAT6_BI[2];
   #htr_2_mod1_flt_cur          :=     #PWR_SPL_STAT6_BI[3];
   #htr_2_mod1_flt_vlt          :=     #PWR_SPL_STAT6_BI[4];
   #htr_2_mod1_flt_save         :=     #PWR_SPL_STAT6_BI[5];
   #htr_2_mod1_flt_rect         :=     #PWR_SPL_STAT6_BI[6];
   #htr_2_mod1_flt_tmp          :=     #PWR_SPL_STAT6_BI[7];

   //---------fault heater 2 modul 2
   #htr_2_mod2_flt_syn_kab      :=     #PWR_SPL_STAT6_BI[8];
   #htr_2_mod2_flt_sys_tmp      :=     #PWR_SPL_STAT6_BI[9];
   #htr_2_mod2_flt_drv          :=     #PWR_SPL_STAT6_BI[10];
   #htr_2_mod2_flt_cur          :=     #PWR_SPL_STAT6_BI[11];
   #htr_2_mod2_flt_vlt          :=     #PWR_SPL_STAT6_BI[12];
   #htr_2_mod2_flt_save         :=     #PWR_SPL_STAT6_BI[13];
   #htr_2_mod2_flt_rect         :=     #PWR_SPL_STAT6_BI[14];
   #htr_2_mod2_flt_tmp          :=     #PWR_SPL_STAT6_BI[15];

   //---------fault heater 2 modul 3
   #flt_htr2_rct_tmp            :=     #PWR_SPL_STAT7_BI[8];                    // heater 2 filter reactor temperature too high 

   #htr_2_mod3_flt_syn_kab      :=     #PWR_SPL_STAT7_BI[0];
   #htr_2_mod3_flt_sys_tmp      :=     #PWR_SPL_STAT7_BI[1];
   #htr_2_mod3_flt_drv          :=     #PWR_SPL_STAT7_BI[2];
   #htr_2_mod3_flt_cur          :=     #PWR_SPL_STAT7_BI[3];
   #htr_2_mod3_flt_vlt          :=     #PWR_SPL_STAT7_BI[4];
   #htr_2_mod3_flt_save         :=     #PWR_SPL_STAT7_BI[5];
   #htr_2_mod3_flt_rect         :=     #PWR_SPL_STAT7_BI[6];
   #htr_2_mod3_flt_tmp          :=     #PWR_SPL_STAT7_BI[7];


   //---------------------------
   //set power to power supply

   "P_BM_PWR_SPL_1_SET_PWR":P := #PWR_SPL_1_SET_PWR; 
   "P_BM_PWR_SPL_2_SET_PWR":P := #PWR_SPL_2_SET_PWR; 


      IF #htr_1_enb THEN                                  
           #PWR_SPL_CTRL.B00_HTR_1_ON   := TRUE;                  // Schalte heater 1 EIN
           #PWR_SPL_1_SET_PWR           := #set_htr_1_pwr;     // Sollwert Leistung

      ELSE
           #PWR_SPL_CTRL.B00_HTR_1_ON   := FALSE;                 // Schalte heater 1 AUS
           #PWR_SPL_1_SET_PWR           := 0.0;                   // Sollwert Leistung 0

      END_IF;

      IF #htr_2_enb THEN                                  
           #PWR_SPL_CTRL.B02_HTR_2_ON   := TRUE;                  // Schalte heater 2 EIN
           #PWR_SPL_2_SET_PWR           := #set_htr_2_pwr;     // Sollwert Leistung

      ELSE
           #PWR_SPL_CTRL.B02_HTR_2_ON   := FALSE;                 // Schalte heater 2 AUS
           #PWR_SPL_2_SET_PWR           := 0.0;                   // Sollwert Leistung 0

      END_IF;
END_FUNCTION_BLOCK

FUNCTION_BLOCK "BM_XT_HDL"   // FB60, SCL
{ S7_Optimized_Access := 'FALSE' }
VERSION : 0.0
// --------------------------------------------------------------------------------
//     program     :   BM_XT_HDL
//     description :   xtal handling
//     name        :   John Wang
//     date        :   15.11.2018
//   
//     revision    :
//     name        :
//     date        :    
//                     (c)PVA CGS GmbH
//     --------------------------------------------------------------------------------
   VAR
      XT_HDL_LFT : "PM_DRV_COMM_LZI950";
      XT_HDL_SW : "PM_DRV_COMM_LZI950";
      xt_hdl_lft_fast : Bool;
      rel_lft_sw_pos_ok : Bool;
      rel_lft_slid_pos_ok : Bool;
      rel_lft_tilt_pos_ok : Bool;
      XT_HDL_SW_STOP : Bool;
      XT_HDL_SW_ERR : Bool;
      XT_HDL_SW_REF : Bool;
      XT_HDL_SW_RUN : Bool;
      XT_HDL_SW_LS_NEG : Bool;
      XT_HDL_SW_LS_POS : Bool;
      XT_HDL_SW_READY : Bool;
      XT_HDL_SW_UP : Bool;
      XT_HDL_SW_REL_REF : Bool;
      XT_HDL_SW_ERROR_CODE : DInt;
      XT_HDL_SW_ACT_POS : Real;
      XT_HDL_SW_ACT_SPEED : Real;
      set_speed : Real;
      op_flt_dly : Int;
      cl_flt_dly : Int;
      xt_hdl_lft_fst_del : Int;
      sw_lock_dly : Int;
      gch_prs_prev : Bool;
      LT_Dummy : Bool;
      KYD_Dummy : Bool;
      rel_man_move : Bool;
      REL_XT_CLP_POS_OK : Bool;
      REL_XT_HDL_SW_IN_OK : Bool;
      REL_XT_HDL_SW_OUT_OK : Bool;
      REL_XT_HDL_SW_DRV : Bool;
      REL_XT_CLP_TILT_POS_OK : Bool;
   END_VAR
BEGIN


       //cystal handling lifting down limit     
        "DV".LS_XT_HDL_LFT_DN_POS  :=  ("DV".LS_XT_HDL_SW_OUT_MAX_POS AND ("DIS".ACT_POS_XT_HDL_LFT < 100.0)) OR
                                    ("DV".LS_XT_HDL_SW_IN_TRP_POS AND ("DIS".ACT_POS_XT_HDL_LFT < "CNF".XT_HDL_LFT_TRP_POS) AND NOT "PDI".LS_HOI_TOOL_INST) OR
                                    ("DV".LS_XT_HDL_SW_IN_TRP_POS AND ("DIS".ACT_POS_XT_HDL_LFT < "CNF".XT_HDL_LFT_TRP_POS) AND "PDI".LS_HOI_TOOL_INST) OR
                                    ("DV".LS_XT_HDL_SW_IN_XT_POS AND ("DIS".ACT_POS_XT_HDL_LFT < "CNF".XT_HDL_LFT_REL_SW_IN)) OR
                                    ("DV".LS_XT_HDL_SW_IN_CRU_POS AND ("DIS".ACT_POS_XT_HDL_LFT < 100.0));
       //cystal handling lifting up limit 
        "DV".LS_XT_HDL_LFT_UP_POS  :=  ("DV".LS_XT_HDL_SW_OUT_MAX_POS AND ("DIS".ACT_POS_XT_HDL_LFT > "CNF".XT_HDL_MAX_UP_POS)) OR    // 2600mm
                                    ("DV".LS_XT_HDL_SW_IN_TRP_POS AND ("DIS".ACT_POS_XT_HDL_LFT > "CNF".XT_ACP_LFT_MID_POS))    OR    // 1500mm
                                    ("DV".LS_XT_HDL_SW_IN_XT_POS AND "LT".LS_XT_TILT_75 AND ("DIS".ACT_POS_XT_HDL_LFT > "CNF".XT_ACP_LFT_UPR_POS)) OR    // 1550mm
                                    ("DV".LS_XT_HDL_SW_IN_XT_POS AND NOT "LT".LS_XT_TILT_75 AND ("DIS".ACT_POS_XT_HDL_LFT > "CNF".XT_HDL_SW_IN_UP_POS)) OR // 1600mm
                                    (("DIS".ACT_POS_XT_HDL_SW>"CNF".XT_HDL_SW_IN_POS) AND ("DIS".ACT_POS_XT_HDL_LFT > "CNF".XT_HDL_LFT_CRU_UP_POS));   // 1490mm

       //cystal handling lifting position limits
        "DV".LS_XT_HDL_LFT_TRP_POS := ABS("DIS".ACT_POS_XT_HDL_LFT-"CNF".XT_HDL_LFT_TRP_POS) < 0.5;   // transport  cart's position 135mm   
        "DV".LS_XT_ACP_LFT_MID_POS := ABS("DIS".ACT_POS_XT_HDL_LFT-"CNF".XT_ACP_LFT_MID_POS) < 0.5;   // acceptance middle position 1500mm  
        "DV".LS_XT_ACP_LFT_LWR_POS := ABS("DIS".ACT_POS_XT_HDL_LFT-"CNF".XT_ACP_LFT_LWR_POS) < 0.5;   // acceptance lower position 1480mm      
        "DV".LS_XT_ACP_LFT_UPR_POS := ABS("DIS".ACT_POS_XT_HDL_LFT-"CNF".XT_ACP_LFT_UPR_POS) < 0.5;   // acceptance upper position 1550mm


       //cystal handling swivel in limit 
        "DV".LS_XT_HDL_SW_IN_POS   := ("DV".LS_XT_HDL_LFT_TRP_POS AND "DV".LS_XT_HDL_SW_IN_TRP_POS) OR   // 53?  
                                   ("DV".LS_XT_HDL_SW_IN_XT_POS AND "DIS".ACT_POS_XT_HDL_LFT>= "CNF".XT_HDL_LFT_REL_SW_IN)  OR   // 143?
                                   ("DV".LS_XT_HDL_SW_IN_CRU_POS AND ("DIS".ACT_POS_XT_HDL_SW>="CNF".XT_HDL_SW_IN_CRU_POS));   // 181?

       //cystal handling swivel out limit
       //DV.LS_XT_HDL_SW_OUT_POS  := (DV.LS_XT_ACP_LFT_UPR_POS AND DV.LS_XT_HDL_SW_IN_TRP_POS) OR   // 45?
       //                              (DV.LS_XT_HDL_SW_OUT_MAX_POS);                              // 10?

       //cystal handling swivel position limits
        "DV".LS_XT_HDL_SW_OUT_MAX_POS := "DIS".ACT_POS_XT_HDL_SW  <= "CNF".XT_HDL_SW_OUT_POS;              // park position 10?  
        "DV".LS_XT_HDL_SW_IN_TRP_POS  := ABS("DIS".ACT_POS_XT_HDL_SW - "CNF".XT_HDL_SW_IN_TRP_POS) < 1.0;  // transport cart's position 53?
        "DV".LS_XT_HDL_SW_IN_XT_POS   := ABS("DIS".ACT_POS_XT_HDL_SW - "CNF".XT_HDL_SW_IN_POS) <1.0;       // position (in) 143?
        "DV".LS_XT_HDL_SW_IN_CRU_POS  := ("DIS".ACT_POS_XT_HDL_SW>= ("CNF".XT_HDL_SW_IN_CRU_POS-0.5));     // position (in) 181?

       //----------------------------------------------------------------------
       // xtal handling lift drive                     
       //----------------------------------------------------------------------
       // controller enable crystal handling lift 
        "PDO".XT_HDL_LFT_ENB := "PDI".EMO AND "PDI".EMS; 

       //xtal handling lift down
        "CM_ITL_IO"(ADR := 65,
             KYD_ON := "KYD".XT_HDL_LFT_DN AND "PDI".MP_ENB_K9,         
             KYD_OFF := NOT "KYD".XT_HDL_LFT_DN OR NOT "PDI".MP_ENB_K9,  
             AUTO := "DV".XT_HDL_SEQ_MOD,  
             DC_ON := "DC".XT_HDL_LFT_DN AND "PDI".MP_ENB_K9, 
             CON1 := "PDI".EMO AND "PDI".EMS,
             CON2 := NOT "FLT".XT_HDL_LFT_ERR,
             CON3 := "SysLog1",  
             CON4 := NOT ("DV".LS_XT_HDL_LFT_DN_POS AND NOT "DV".MP_SERVICE),    
             CON5 := #rel_lft_sw_pos_ok  OR "DV".MP_SERVICE,   
             CON6 := #rel_lft_slid_pos_ok,                                              
             CON7 := #rel_lft_tilt_pos_ok,    
             CON8 := "SysLog1",   
             ITL_OUT := "STA_ITL_CAUSE",
             LT_OUT := "LT".XT_HDL_LFT_DN);     

        "LT".XT_HDL_LFT_DN_REL  :=          "PDI".EMO AND "PDI".EMS
                                 AND NOT "FLT".XT_HDL_LFT_ERR
                                 AND NOT ("DV".LS_XT_HDL_LFT_DN_POS  AND NOT "DV".MP_SERVICE) 
                                 AND     (#rel_lft_sw_pos_ok  OR "DV".MP_SERVICE) 
                                 AND     #rel_lft_slid_pos_ok 
                                 AND     #rel_lft_tilt_pos_ok;  

       // ----------------xtal handling lift up ---------------------------------  
        "CM_ITL_IO"(ADR := 66,
             KYD_ON := "KYD".XT_HDL_LFT_UP AND "PDI".MP_ENB_K9,
             KYD_OFF := NOT "KYD".XT_HDL_LFT_UP OR NOT "PDI".MP_ENB_K9,
             AUTO := "DV".XT_HDL_SEQ_MOD,  
             DC_ON := "DC".XT_HDL_LFT_UP AND "PDI".MP_ENB_K9, 
             CON1 := "PDI".EMO AND "PDI".EMS,
             CON2 := NOT "FLT".XT_HDL_LFT_ERR,
             CON3 := "SysLog1",   
             CON4 := NOT "DV".LS_XT_HDL_LFT_UP_POS OR "DV".MP_SERVICE, 
             CON5 := #rel_lft_sw_pos_ok OR "DV".MP_SERVICE,   
             CON6 := #rel_lft_slid_pos_ok OR "DV".MP_SERVICE,                     
             CON7 := #rel_lft_tilt_pos_ok,    
             CON8 := "SysLog1",   
             ITL_OUT:= "STA_ITL_CAUSE",
             LT_OUT := "LT".XT_HDL_LFT_UP);


        "LT".XT_HDL_LFT_UP_REL   :=         "PDI".EMO AND "PDI".EMS
                                 AND NOT "FLT".XT_HDL_LFT_ERR
                                 AND NOT ("DV".LS_XT_HDL_LFT_UP_POS  AND NOT "DV".MP_SERVICE)
                                 AND     (#rel_lft_sw_pos_ok OR "DV".MP_SERVICE) 
                                 AND     #rel_lft_slid_pos_ok 
                                 AND     #rel_lft_tilt_pos_ok;                                                    


        #rel_lft_sw_pos_ok   := "DV".LS_XT_HDL_SW_OUT_MAX_POS OR "DV".LS_XT_HDL_SW_IN_TRP_POS OR "DV".LS_XT_HDL_SW_IN_XT_POS OR "DV".LS_XT_HDL_SW_IN_CRU_POS; 
        #rel_lft_slid_pos_ok := ("LT".LS_XT_SLID_BW AND ((NOT "DV".LS_XT_HDL_SW_IN_TRP_POS OR ("DIS".ACT_POS_XT_HDL_LFT>620.0)) OR NOT "PDI".LS_XT_CLP_CON)) OR "LT".LS_XT_SLID_FW; // OR NOT PDI.LS_XT_CLP_CON; 
        #rel_lft_tilt_pos_ok := "LT".LS_XT_TILT_90 OR "LT".LS_XT_TILT_75 OR NOT "PDI".LS_XT_CLP_CON; 

       // Set speed  
        IF "DV".XT_HDL_SEQ_MOD THEN
          #xt_hdl_lft_fast := ("KYD".XT_HDL_LFT_FAST AND NOT "DV".XT_HDL_SEQ_MOD) 
                          OR ("DC".XT_HDL_LFT_FAST AND "DV".XT_HDL_SEQ_MOD);
        ELSE
          IF "LT".XT_HDL_LFT_UP OR "LT".XT_HDL_LFT_DN THEN
             IF #xt_hdl_lft_fst_del<5 THEN
                #xt_hdl_lft_fst_del := #xt_hdl_lft_fst_del + 1;
             ELSE
                #xt_hdl_lft_fast :=  "KYD".XT_HDL_LFT_FAST OR
                                   ("DV".LS_XT_HDL_SW_OUT_MAX_POS AND ("DIS".ACT_POS_XT_HDL_LFT>20.0) AND ("DIS".ACT_POS_XT_HDL_LFT<2200.0)) OR
                                   ("DV".LS_XT_HDL_SW_IN_TRP_POS AND ("DIS".ACT_POS_XT_HDL_LFT>620.0) AND ("DIS".ACT_POS_XT_HDL_LFT<1700.0)) OR
                                   ("DV".LS_XT_HDL_SW_IN_XT_POS AND ("DIS".ACT_POS_XT_HDL_LFT>20.0) AND ("DIS".ACT_POS_XT_HDL_LFT<1700.0) AND "SysLog0");
             END_IF;   
          ELSE
             #xt_hdl_lft_fst_del := 0;
             #xt_hdl_lft_fast := False;  
          END_IF;                       
        END_IF;   

        IF "LT".XT_HDL_LFT_UP THEN 
          IF #xt_hdl_lft_fast THEN
             #set_speed  := "CNF_XT_HDL_LFT_LZ950".MAX_SPEED;  // lift up fast 
          ELSE   
             #set_speed  := "CNF_XT_HDL_LFT_LZ950".SEL_SPEED;  // lift up 
          END_IF;
        END_IF;       
        IF "LT".XT_HDL_LFT_DN THEN 
          IF #xt_hdl_lft_fast THEN
             #set_speed  := -"CNF_XT_HDL_LFT_LZ950".MAX_SPEED;  // lift dn fast 
          ELSE   
             #set_speed  := -"CNF_XT_HDL_LFT_LZ950".SEL_SPEED;  // lift dn 
          END_IF;
        END_IF;       
        IF NOT "LT".XT_HDL_LFT_UP AND NOT "LT".XT_HDL_LFT_DN THEN 
          #set_speed  := 0.0; 
        END_IF;


       // Release reference run
        "LT".XT_HDL_LFT_REF_RUN := (("LT".XT_HDL_LFT_REF_RUN OR "KYD".XT_HDL_LFT_REF_START) 
                              AND NOT "LT".XT_HDL_LFT_REF_DONE) 
                              AND NOT "KYD".XT_HDL_LFT_REF_RES 
                              AND NOT "APC".AUTOMATIC AND ("APC".STATUS=0) 
                              AND NOT "DV".XT_HDL_SEQ_MOD 
                              AND NOT "PDI".LS_XT_CLP_CON
                              AND NOT "DV".EMG_STOP
                              AND NOT "FLT".DRV_XT_LFT_RUN_FLT
                              AND NOT #XT_HDL_LFT.Error;


        "LT".XT_HDL_LFT_REF_DONE := #XT_HDL_LFT.Ref_Done OR "SY".SIM_ON;                     

        #XT_HDL_LFT(Enable        := INT_TO_BOOL("CNF_XT_HDL_LFT_LZ950".CTRL_ACTIV) AND ("LT".XT_HDL_LFT_UP OR "LT".XT_HDL_LFT_DN OR "LT".XT_HDL_LFT_REF_RUN), 
                   Pro_start     := "LT".XT_HDL_LFT_UP OR "LT".XT_HDL_LFT_DN,   
                   Speed_ext_ovr := TRUE,   
                   Ref_Start     := "LT".XT_HDL_LFT_REF_RUN,
                   Ref_reset     := "KYD".XT_HDL_LFT_REF_RES AND NOT "APC".AUTOMATIC AND ("APC".STATUS=0) AND NOT "DV".XT_HDL_SEQ_MOD AND NOT "PDI".LS_XT_CLP_CON,
                   Reset_error   := "KYD".XT_HDL_LFT_TRIP_RES,
                   Stop          := NOT "LT".XT_HDL_LFT_UP AND NOT "LT".XT_HDL_LFT_DN,
                   Profil        := "CNF_XT_HDL_LFT_LZ950".Profil,
                   PM_ADR_E      := INT_TO_WORD("CNF_XT_HDL_LFT_LZ950".PE_ADR),                                    
                   PM_ADR_A      := INT_TO_WORD("CNF_XT_HDL_LFT_LZ950".PA_ADR),                
                   Units_per_rev := "CNF_XT_HDL_LFT_LZ950".UNITS_PER_REV,                       
                   Gear_ratio    := "CNF_XT_HDL_LFT_LZ950".FEED_CONST,
                   Set_vel       := #set_speed); 


       //actual motor values
       //---------------------
        IF NOT "SY".SIM_ON THEN
          "AV".XT_HDL_LFT_ACT_POS  := #XT_HDL_LFT.Act_pos; 
        END_IF;
        "DIS".ACT_POS_XT_HDL_LFT  := "AV".XT_HDL_LFT_ACT_POS;   

       //actual fault
       //---------------------
        "DIS".XT_HDL_LFT_ERR_CODE := #XT_HDL_LFT.Error_code;        // Fehlernummer Umrichter
        "FLT".XT_HDL_LFT_ERR      := #XT_HDL_LFT.Error;             // Fehlerbit Umrichter
        "FLT".XT_HDL_LFT_POS_REF  := NOT "LT".XT_HDL_LFT_REF_DONE;   // Antrieb nicht referenziert
        "FLT".XT_HDL_LFT_SLS      := #XT_HDL_LFT.LS_neg OR #XT_HDL_LFT.LS_pos;  // Fehler Sicherheitsendschalter

       //----------------------------------------------------------------------
       // xtal handling swiveling drive           
       //----------------------------------------------------------------------
       // controller enable crystal handling swivel 
        "PDO".XT_HDL_SW_ENB  := "PDI".EMO AND "PDI".EMS;  

       // xtal handling lift swivel out
        "CM_ITL_IO"(ADR := 67,
             KYD_ON := "KYD".XT_HDL_SW_OUT AND "PDI".MP_ENB_K9 AND #REL_XT_HDL_SW_DRV,
             KYD_OFF := NOT "KYD".XT_HDL_SW_OUT OR NOT "PDI".MP_ENB_K9,
             AUTO  := "DV".XT_HDL_SEQ_MOD, 
             DC_ON := "DC".XT_HDL_SW_OUT AND "PDI".MP_ENB_K9,
             CON1 := "PDI".EMO AND "PDI".EMS,
             CON2 := NOT "FLT".XT_HDL_SW_ERR,
             CON3 := "PDI".LS_XT_HDL_SW_UNLOCK AND NOT "PDI".LS_XT_HDL_SW_LOCK, 
             CON4 := #REL_XT_HDL_SW_OUT_OK OR "DV".MP_SERVICE,   
             CON5 := NOT "DV".LS_XT_HDL_SW_OUT_MAX_POS OR "DV".MP_SERVICE,   
             CON6 := "SysLog1",                     
             CON7 := "SysLog1",    
             CON8 := "SysLog1",   
             ITL_OUT := "STA_ITL_CAUSE",
             LT_OUT := "LT".XT_HDL_SW_OUT); 

         "LT".LS_XT_HDL_SW_OUT  := "DV".LS_XT_HDL_SW_OUT_MAX_POS;
         "LT".XT_HDL_SW_OUT_REL := "PDI".EMO AND "PDI".EMS
                               AND NOT "FLT".XT_HDL_SW_ERR
                               //AND PDI.LS_XT_HDL_SW_UNLOCK AND NOT PDI.LS_XT_HDL_SW_LOCK 
                               AND (#REL_XT_HDL_SW_OUT_OK OR "DV".MP_SERVICE)   
                               AND (NOT "DV".LS_XT_HDL_SW_OUT_MAX_POS OR "DV".MP_SERVICE);

         #REL_XT_HDL_SW_OUT_OK := (NOT "PDI".LS_XT_SLID_BW OR NOT "PDI".LS_XT_CLP_CON) AND ("DIS".ACT_POS_XT_HDL_LFT>1160.0);

